  Call Extruder 0.1366
  MoveL (T14464) to (106.09, 106.63, 16.1) mm, rotated rx 180 ry 0 rz -180 deg; joints [1.434, 67.125, -29.697, 2.359, -37.451, -1.873]
  Call Extruder 0.01306
  MoveL (T14465) to (106.44, 106.98, 16.1) mm, rotated rx 180 ry 0 rz -180 deg; joints [1.434, 67.125, -29.697, 2.359, -37.451, -1.873]
  Call Extruder 0.12393
  MoveL (T14466) to (111.15, 106.98, 16.1) mm, rotated rx 180 ry 0 rz -180 deg; joints [1.434, 67.125, -29.697, 2.359, -37.451, -1.873]
  Set speed (150.0 mm/s)
  MoveL (T14467) to (112.51, 106.28, 16.1) mm, rotated rx 180 ry 0 rz -180 deg; joints [1.744, 66.421, -28.373, 2.828, -38.082, -2.227]
  Set speed (25.0 mm/s)
  MoveL (T14468) to (112.51, 106.28, 16.1) mm, rotated rx 180 ry 0 rz -180 deg; joints [1.744, 66.421, -28.373, 2.828, -38.082, -2.227]
  Call Extruder 0.22808
  MoveL (T14469) to (121.19, 106.28, 16.1) mm, rotated rx 180 ry 0 rz -180 deg; joints [1.744, 66.421, -28.373, 2.828, -38.082, -2.227]
  Call Extruder 0.00923
  MoveL (T14470) to (121.19, 106.63, 16.1) mm, rotated rx 180 ry 0 rz -180 deg; joints [1.681, 66.417, -28.365, 2.726, -38.083, -2.146]
  Call Extruder 0.21306
  MoveL (T14471) to (113.08, 106.63, 16.1) mm, rotated rx 180 ry 0 rz -180 deg; joints [1.681, 66.417, -28.365, 2.726, -38.083, -2.146]
  Call Extruder 0.01306
  MoveL (T14472) to (113.43, 106.98, 16.1) mm, rotated rx 180 ry 0 rz -180 deg; joints [1.681, 66.417, -28.365, 2.726, -38.083, -2.146]
  Call Extruder 0.20382
  MoveL (T14473) to (121.19, 106.98, 16.1) mm, rotated rx 180 ry 0 rz -180 deg; joints [1.436, 66.973, -29.411, 2.354, -37.585, -1.866]
  Call Extruder 0.00923
  MoveL (T14474) to (121.19, 107.33, 16.1) mm, rotated rx 180 ry 0 rz -180 deg; joints [1.436, 66.973, -29.411, 2.354, -37.585, -1.866]
  Call Extruder 0.09038
  MoveL (T14475) to (117.75, 107.33, 16.1) mm, rotated rx 180 ry 0 rz -180 deg; joints [1.436, 66.973, -29.411, 2.354, -37.585, -1.866]
  Call Extruder 0.00923
  MoveL (T14476) to (117.75, 107.68, 16.1) mm, rotated rx 180 ry 0 rz -180 deg; joints [1.436, 66.973, -29.411, 2.354, -37.585, -1.866]
  Call Extruder 0.09038
  MoveL (T14477) to (121.19, 107.68, 16.1) mm, rotated rx 180 ry 0 rz -180 deg; joints [1.437, 66.821, -29.126, 2.35, -37.719, -1.859]
  Call Extruder 0.00923
  MoveL (T14478) to (121.19, 108.03, 16.1) mm, rotated rx 180 ry 0 rz -180 deg; joints [1.437, 66.821, -29.126, 2.35, -37.719, -1.859]
  Call Extruder 0.09039
  MoveL (T14479) to (117.75, 108.03, 16.1) mm, rotated rx 180 ry 0 rz -180 deg; joints [1.437, 66.821, -29.126, 2.35, -37.719, -1.859]
  Call Extruder 0.00923
  MoveL (T14480) to (117.75, 108.38, 16.1) mm, rotated rx 180 ry 0 rz -180 deg; joints [1.437, 66.821, -29.126, 2.35, -37.719, -1.859]
  Call Extruder 0.09039
  MoveL (T14481) to (121.19, 108.38, 16.1) mm, rotated rx 180 ry 0 rz -180 deg; joints [1.618, 66.412, -28.357, 2.624, -38.085, -2.066]
  Call Extruder 0.00923
  MoveL (T14482) to (121.19, 108.73, 16.1) mm, rotated rx 180 ry 0 rz -180 deg; joints [1.618, 66.412, -28.357, 2.624, -38.085, -2.066]
  Call Extruder 0.0904
  MoveL (T14483) to (117.75, 108.73, 16.1) mm, rotated rx 180 ry 0 rz -180 deg; joints [1.618, 66.412, -28.357, 2.624, -38.085, -2.066]
  Call Extruder 0.00923
  MoveL (T14484) to (117.75, 109.09, 16.1) mm, rotated rx 180 ry 0 rz -180 deg; joints [1.555, 66.408, -28.349, 2.522, -38.086, -1.985]
  Call Extruder 0.0904
  MoveL (T14485) to (121.19, 109.09, 16.1) mm, rotated rx 180 ry 0 rz -180 deg; joints [1.555, 66.408, -28.349, 2.522, -38.086, -1.985]
  Call Extruder 0.00923
  MoveL (T14486) to (121.19, 109.44, 16.1) mm, rotated rx 180 ry 0 rz -180 deg; joints [1.555, 66.408, -28.349, 2.522, -38.086, -1.985]
  Call Extruder 0.0904
  MoveL (T14487) to (117.75, 109.44, 16.1) mm, rotated rx 180 ry 0 rz -180 deg; joints [1.439, 66.67, -28.842, 2.345, -37.851, -1.852]
  Call Extruder 0.00923
  MoveL (T14488) to (117.75, 109.79, 16.1) mm, rotated rx 180 ry 0 rz -180 deg; joints [1.439, 66.67, -28.842, 2.345, -37.851, -1.852]
  Call Extruder 0.09041
  MoveL (T14489) to (121.19, 109.79, 16.1) mm, rotated rx 180 ry 0 rz -180 deg; joints [1.439, 66.67, -28.842, 2.345, -37.851, -1.852]
  Call Extruder 0.00923
  MoveL (T14490) to (121.19, 110.14, 16.1) mm, rotated rx 180 ry 0 rz -180 deg; joints [1.44, 66.521, -28.56, 2.341, -37.983, -1.845]
  Call Extruder 0.09041
  MoveL (T14491) to (117.75, 110.14, 16.1) mm, rotated rx 180 ry 0 rz -180 deg; joints [1.44, 66.521, -28.56, 2.341, -37.983, -1.845]
  Call Extruder 0.00268
  MoveL (T14492) to (117.75, 110.24, 16.1) mm, rotated rx 180 ry 0 rz -180 deg; joints [1.44, 66.521, -28.56, 2.341, -37.983, -1.845]
  Call Extruder 0.00927
  MoveL (T14493) to (118, 110.49, 16.1) mm, rotated rx 180 ry 0 rz -180 deg; joints [1.512, 66.359, -28.256, 2.45, -38.128, -1.928]
  Call Extruder 0.08386
  MoveL (T14494) to (121.19, 110.49, 16.1) mm, rotated rx 180 ry 0 rz -180 deg; joints [1.512, 66.359, -28.256, 2.45, -38.128, -1.928]
  Call Extruder 0.00923
  MoveL (T14495) to (121.19, 110.84, 16.1) mm, rotated rx 180 ry 0 rz -180 deg; joints [1.512, 66.359, -28.256, 2.45, -38.128, -1.928]
  Call Extruder 0.07462
  MoveL (T14496) to (118.35, 110.84, 16.1) mm, rotated rx 180 ry 0 rz -180 deg; joints [1.512, 66.359, -28.256, 2.45, -38.128, -1.928]
  Call Extruder 0.01306
  MoveL (T14497) to (118.7, 111.19, 16.1) mm, rotated rx 180 ry 0 rz -180 deg; joints [1.512, 66.359, -28.256, 2.45, -38.128, -1.928]
  Call Extruder 0.06539
  MoveL (T14498) to (121.19, 111.19, 16.1) mm, rotated rx 180 ry 0 rz -180 deg; joints [1.512, 66.359, -28.256, 2.45, -38.128, -1.928]
  Call Extruder 0.00923
  MoveL (T14499) to (121.19, 111.55, 16.1) mm, rotated rx 180 ry 0 rz -180 deg; joints [1.512, 66.359, -28.256, 2.45, -38.128, -1.928]
  Call Extruder 0.05615
  MoveL (T14500) to (119.05, 111.55, 16.1) mm, rotated rx 180 ry 0 rz -180 deg; joints [1.512, 66.359, -28.256, 2.45, -38.128, -1.928]
  Call Extruder 0.01306
  MoveL (T14501) to (119.4, 111.9, 16.1) mm, rotated rx 180 ry 0 rz -180 deg; joints [1.512, 66.359, -28.256, 2.45, -38.128, -1.928]
  Call Extruder 0.05101
  MoveL (T14502) to (121.34, 111.9, 16.1) mm, rotated rx 180 ry 0 rz -180 deg; joints [1.512, 66.359, -28.256, 2.45, -38.128, -1.928]
  Set speed (45.0 mm/s)
  Call Extruder -1.6
  MoveL (T14503) to (121.34, 111.9, 16.1) mm, rotated rx 180 ry 0 rz -180 deg; joints [1.44, 66.521, -28.56, 2.341, -37.983, -1.845]
  Set speed (120.0 mm/s)
  MoveL (T14504) to (121.34, 111.9, 16.1) mm, rotated rx 180 ry 0 rz -180 deg; joints [1.44, 66.521, -28.56, 2.341, -37.983, -1.845]
  Call Extruder -0.38
  MoveL (T14505) to (120.28, 111.9, 16.1) mm, rotated rx 180 ry 0 rz -180 deg; joints [1.44, 66.521, -28.56, 2.341, -37.983, -1.845]
  Set speed (45.0 mm/s)
  Call Extruder -0.02
  MoveL (T14506) to (120.28, 111.9, 16.1) mm, rotated rx 180 ry 0 rz -180 deg; joints [1.44, 66.521, -28.56, 2.341, -37.983, -1.845]
  Set speed (150.0 mm/s)
  MoveL (T14507) to (120.28, 111.9, 18.1) mm, rotated rx 180 ry 0 rz -180 deg; joints [1.44, 66.559, -28.633, 2.342, -37.949, -1.847]
  MoveL (T14508) to (120.87, 104.13, 18.1) mm, rotated rx 180 ry 0 rz -180 deg; joints [1.44, 66.559, -28.633, 2.342, -37.949, -1.847]
  MoveL (T14509) to (120.87, 104.13, 16.1) mm, rotated rx 180 ry 0 rz -180 deg; joints [1.44, 66.559, -28.633, 2.342, -37.949, -1.847]
  Set speed (40.0 mm/s)
  Call Extruder 2.0
  MoveL (T14510) to (120.87, 104.13, 16.1) mm, rotated rx 180 ry 0 rz -180 deg; joints [1.44, 66.559, -28.633, 2.342, -37.949, -1.847]
  Set speed (50.0 mm/s)
  MoveL (T14511) to (120.87, 104.13, 16.1) mm, rotated rx 180 ry 0 rz -180 deg; joints [1.44, 66.559, -28.633, 2.342, -37.949, -1.847]
  Call Extruder 0.01219
  MoveL (T14512) to (121.16, 103.84, 16.1) mm, rotated rx 180 ry 0 rz -180 deg; joints [1.44, 66.559, -28.633, 2.342, -37.949, -1.847]
  Set speed (45.0 mm/s)
  Call Extruder -1.6
  MoveL (T14513) to (121.16, 103.84, 16.1) mm, rotated rx 180 ry 0 rz -180 deg; joints [1.44, 66.321, -28.593, 2.352, -37.752, -1.86]
  Set speed (120.0 mm/s)
  MoveL (T14514) to (121.16, 103.84, 16.1) mm, rotated rx 180 ry 0 rz -180 deg; joints [1.407, 66.288, -28.531, 2.298, -37.78, -1.816]
  Call Extruder -0.14257
  MoveL (T14515) to (120.87, 104.13, 16.1) mm, rotated rx 180 ry 0 rz -180 deg; joints [1.407, 66.502, -28.567, 2.288, -37.958, -1.805]
  Set speed (45.0 mm/s)
  Call Extruder -0.25743
  MoveL (T14516) to (120.87, 104.13, 16.1) mm, rotated rx 180 ry 0 rz -180 deg; joints [1.407, 66.502, -28.567, 2.288, -37.958, -1.805]
  Set speed (150.0 mm/s)
  MoveL (T14517) to (120.87, 104.13, 18.1) mm, rotated rx 180 ry 0 rz -180 deg; joints [1.407, 66.502, -28.567, 2.288, -37.958, -1.805]
  MoveL (T14518) to (104.34, 103.54, 18.1) mm, rotated rx 180 ry 0 rz -180 deg; joints [1.407, 66.502, -28.567, 2.288, -37.958, -1.805]
  MoveL (T14519) to (104.34, 103.54, 16.3) mm, rotated rx 180 ry 0 rz -180 deg; joints [1.407, 66.502, -28.567, 2.288, -37.958, -1.805]
  Set speed (40.0 mm/s)
  Call Extruder 2.0
  MoveL (T14520) to (104.34, 103.54, 16.3) mm, rotated rx 180 ry 0 rz -180 deg; joints [1.407, 66.502, -28.567, 2.288, -37.958, -1.805]
  Call Extruder 0.52159
  MoveL (T14521) to (121.46, 103.54, 16.3) mm, rotated rx 180 ry 0 rz -180 deg; joints [1.407, 66.502, -28.567, 2.288, -37.958, -1.805]
  Call Extruder 0.54596
  MoveL (T14522) to (121.46, 121.46, 16.3) mm, rotated rx 180 ry 0 rz -180 deg; joints [1.363, 71.341, -37.668, 2.458, -33.696, -2.045]
  Call Extruder 0.54596
  MoveL (T14523) to (103.54, 121.46, 16.3) mm, rotated rx 180 ry 0 rz -180 deg; joints [1.363, 71.341, -37.668, 2.458, -33.696, -2.045]
  Call Extruder 0.54596
  MoveL (T14524) to (103.54, 103.54, 16.3) mm, rotated rx 180 ry 0 rz -180 deg; joints [1.363, 71.341, -37.668, 2.458, -33.696, -2.045]
  Call Extruder 0.02254
  MoveL (T14525) to (104.28, 103.54, 16.3) mm, rotated rx 180 ry 0 rz -180 deg; joints [3.241, 71.568, -38.096, 5.863, -33.61, -4.888]
  Set speed (150.0 mm/s)
  MoveL (T14526) to (103.53, 103.13, 16.3) mm, rotated rx 180 ry 0 rz -180 deg; joints [3.241, 71.568, -38.096, 5.863, -33.61, -4.888]
  Set speed (40.0 mm/s)
  MoveL (T14527) to (103.53, 103.13, 16.3) mm, rotated rx 180 ry 0 rz -180 deg; joints [3.241, 71.568, -38.096, 5.863, -33.61, -4.888]
  Call Extruder 0.55858
  MoveL (T14528) to (121.87, 103.13, 16.3) mm, rotated rx 180 ry 0 rz -180 deg; joints [3.241, 71.568, -38.096, 5.863, -33.61, -4.888]
  Call Extruder 0.57077
  MoveL (T14529) to (121.87, 121.87, 16.3) mm, rotated rx 180 ry 0 rz -180 deg; joints [3.351, 66.488, -28.54, 5.439, -38.073, -4.287]
  Call Extruder 0.57077
  MoveL (T14530) to (103.13, 121.87, 16.3) mm, rotated rx 180 ry 0 rz -180 deg; joints [3.351, 66.488, -28.54, 5.439, -38.073, -4.287]
  Call Extruder 0.57077
  MoveL (T14531) to (103.13, 103.13, 16.3) mm, rotated rx 180 ry 0 rz -180 deg; joints [3.351, 66.488, -28.54, 5.439, -38.073, -4.287]
  Call Extruder 0.01036
  MoveL (T14532) to (103.47, 103.13, 16.3) mm, rotated rx 180 ry 0 rz -180 deg; joints [1.409, 66.297, -28.181, 2.283, -38.138, -1.796]
  Set speed (150.0 mm/s)
  MoveL (T14533) to (102.72, 102.81, 16.3) mm, rotated rx 180 ry 0 rz -180 deg; joints [1.409, 66.297, -28.181, 2.283, -38.138, -1.796]
  Set speed (25.0 mm/s)
  MoveL (T14534) to (102.72, 102.81, 16.3) mm, rotated rx 180 ry 0 rz -180 deg; joints [1.409, 66.297, -28.181, 2.283, -38.138, -1.796]
  Call Extruder 0.00259
  MoveL (T14535) to (102.72, 102.72, 16.3) mm, rotated rx 180 ry 0 rz -180 deg; joints [1.407, 66.487, -28.538, 2.288, -37.971, -1.804]
  Call Extruder 0.59557
  MoveL (T14536) to (122.28, 102.72, 16.3) mm, rotated rx 180 ry 0 rz -180 deg; joints [1.407, 66.487, -28.538, 2.288, -37.971, -1.804]
  Call Extruder 0.59557
  MoveL (T14537) to (122.28, 122.28, 16.3) mm, rotated rx 180 ry 0 rz -180 deg; joints [1.407, 66.487, -28.538, 2.288, -37.971, -1.804]
  Call Extruder 0.59557
  MoveL (T14538) to (102.72, 122.28, 16.3) mm, rotated rx 180 ry 0 rz -180 deg; joints [1.365, 66.293, -28.173, 2.211, -38.141, -1.739]
  Call Extruder 0.59115
  MoveL (T14539) to (102.72, 102.87, 16.3) mm, rotated rx 180 ry 0 rz -180 deg; joints [1.365, 66.293, -28.173, 2.211, -38.141, -1.739]
  Set speed (150.0 mm/s)
  MoveL (T14540) to (102.78, 102.75, 16.3) mm, rotated rx 180 ry 0 rz -180 deg; joints [1.365, 66.293, -28.173, 2.211, -38.141, -1.739]
  Set speed (45.0 mm/s)
  Call Extruder -1.6
  MoveL (T14541) to (102.78, 102.75, 16.3) mm, rotated rx 180 ry 0 rz -180 deg; joints [1.365, 66.293, -28.173, 2.211, -38.141, -1.739]
  Set speed (120.0 mm/s)
  MoveL (T14542) to (102.78, 102.75, 16.3) mm, rotated rx 180 ry 0 rz -180 deg; joints [1.365, 66.293, -28.173, 2.211, -38.141, -1.739]
  Call Extruder -0.05166
  MoveL (T14543) to (102.72, 102.72, 16.3) mm, rotated rx 180 ry 0 rz -180 deg; joints [1.365, 66.293, -28.173, 2.211, -38.141, -1.739]
  Call Extruder -0.32834
  MoveL (T14544) to (103.65, 102.72, 16.3) mm, rotated rx 180 ry 0 rz -180 deg; joints [1.319, 71.466, -37.904, 2.386, -33.585, -1.988]
  Set speed (45.0 mm/s)
  Call Extruder -0.02
  MoveL (T14545) to (103.65, 102.72, 16.3) mm, rotated rx 180 ry 0 rz -180 deg; joints [1.319, 71.466, -37.904, 2.386, -33.585, -1.988]
  Set speed (150.0 mm/s)
  MoveL (T14546) to (103.65, 102.72, 18.3) mm, rotated rx 180 ry 0 rz -180 deg; joints [3.282, 71.704, -38.353, 5.954, -33.494, -4.971]
  MoveL (T14547) to (103.84, 106.29, 18.3) mm, rotated rx 180 ry 0 rz -180 deg; joints [3.282, 71.704, -38.353, 5.954, -33.494, -4.971]
  MoveL (T14548) to (103.84, 106.29, 16.3) mm, rotated rx 180 ry 0 rz -180 deg; joints [3.398, 66.39, -28.356, 5.504, -38.163, -4.333]
  Set speed (40.0 mm/s)
  Call Extruder 2.0
  MoveL (T14549) to (103.84, 106.29, 16.3) mm, rotated rx 180 ry 0 rz -180 deg; joints [1.366, 66.191, -27.981, 2.208, -38.23, -1.735]
  Set speed (42.3 mm/s)
  MoveL (T14550) to (103.84, 106.29, 16.3) mm, rotated rx 180 ry 0 rz -180 deg; joints [1.366, 66.191, -27.981, 2.208, -38.23, -1.735]
  Call Extruder 0.07441
  MoveL (T14551) to (103.84, 103.84, 16.3) mm, rotated rx 180 ry 0 rz -180 deg; joints [1.365, 66.278, -28.144, 2.211, -38.154, -1.739]
  Call Extruder 0.0111
  MoveL (T14552) to (104.1, 104.1, 16.3) mm, rotated rx 180 ry 0 rz -180 deg; joints [1.365, 66.278, -28.144, 2.211, -38.154, -1.739]
  Call Extruder 0.05294
  MoveL (T14553) to (104.1, 105.84, 16.3) mm, rotated rx 180 ry 0 rz -180 deg; joints [1.365, 66.278, -28.144, 2.211, -38.154, -1.739]
  Call Extruder 0.00661
  MoveL (T14554) to (104.18, 106.04, 16.3) mm, rotated rx 180 ry 0 rz -180 deg; joints [1.332, 66.086, -27.783, 2.149, -38.322, -1.686]
  Call Extruder 0.02065
  MoveL (T14555) to (104.66, 106.52, 16.3) mm, rotated rx 180 ry 0 rz -180 deg; joints [1.332, 66.086, -27.783, 2.149, -38.322, -1.686]
  Call Extruder 0.03528
  MoveL (T14556) to (103.84, 107.34, 16.3) mm, rotated rx 180 ry 0 rz -180 deg; joints [1.332, 66.086, -27.783, 2.149, -38.322, -1.686]
  Call Extruder 0.03385
  MoveL (T14557) to (103.84, 108.45, 16.3) mm, rotated rx 180 ry 0 rz -180 deg; joints [1.332, 66.086, -27.783, 2.149, -38.322, -1.686]
  Call Extruder 0.54738
  MoveL (T14558) to (116.55, 121.16, 16.3) mm, rotated rx 180 ry 0 rz -180 deg; joints [1.323, 66.085, -27.782, 2.134, -38.322, -1.675]
  Call Extruder 0.03385
  MoveL (T14559) to (117.66, 121.16, 16.3) mm, rotated rx 180 ry 0 rz -180 deg; joints [1.323, 66.085, -27.782, 2.134, -38.322, -1.675]
  Call Extruder 0.05922
  MoveL (T14560) to (119.04, 119.78, 16.3) mm, rotated rx 180 ry 0 rz -180 deg; joints [1.323, 66.085, -27.782, 2.134, -38.322, -1.675]
  Call Extruder 0.00883
  MoveL (T14561) to (119.24, 119.99, 16.3) mm, rotated rx 180 ry 0 rz -180 deg; joints [1.276, 71.591, -38.14, 2.314, -33.472, -1.93]
  Call Extruder 0.02274
  MoveL (T14562) to (119.99, 119.99, 16.3) mm, rotated rx 180 ry 0 rz -180 deg; joints [1.276, 71.591, -38.14, 2.314, -33.472, -1.93]
  Call Extruder 0.05034
  MoveL (T14563) to (121.16, 121.16, 16.3) mm, rotated rx 180 ry 0 rz -180 deg; joints [3.322, 71.842, -38.612, 6.046, -33.377, -5.054]
  Call Extruder 0.07441
  MoveL (T14564) to (118.71, 121.16, 16.3) mm, rotated rx 180 ry 0 rz -180 deg; joints [3.322, 71.842, -38.612, 6.046, -33.377, -5.054]
  Set speed (45.0 mm/s)
  Call Extruder -1.6
  MoveL (T14565) to (118.71, 121.16, 16.3) mm, rotated rx 180 ry 0 rz -180 deg; joints [3.322, 71.842, -38.612, 6.046, -33.377, -5.054]
  Set speed (120.0 mm/s)
  MoveL (T14566) to (118.71, 121.16, 16.3) mm, rotated rx 180 ry 0 rz -180 deg; joints [3.445, 66.292, -28.172, 5.569, -38.252, -4.379]
  Call Extruder -0.38
  MoveL (T14567) to (119.78, 121.16, 16.3) mm, rotated rx 180 ry 0 rz -180 deg; joints [3.445, 66.292, -28.172, 5.569, -38.252, -4.379]
  Set speed (45.0 mm/s)
  Call Extruder -0.02
  MoveL (T14568) to (119.78, 121.16, 16.3) mm, rotated rx 180 ry 0 rz -180 deg; joints [3.445, 66.292, -28.172, 5.569, -38.252, -4.379]
  Set speed (150.0 mm/s)
  MoveL (T14569) to (119.78, 121.16, 18.3) mm, rotated rx 180 ry 0 rz -180 deg; joints [1.339, 66.086, -27.784, 2.16, -38.322, -1.695]
  MoveL (T14570) to (117.37, 115.49, 18.3) mm, rotated rx 180 ry 0 rz -180 deg; joints [1.339, 66.086, -27.784, 2.16, -38.322, -1.695]
  MoveL (T14571) to (117.37, 115.49, 16.3) mm, rotated rx 180 ry 0 rz -180 deg; joints [1.339, 66.086, -27.784, 2.16, -38.322, -1.695]
  Set speed (40.0 mm/s)
  Call Extruder 2.0
  MoveL (T14572) to (117.37, 115.49, 16.3) mm, rotated rx 180 ry 0 rz -180 deg; joints [1.339, 66.086, -27.784, 2.16, -38.322, -1.695]
  Set speed (42.3 mm/s)
  MoveL (T14573) to (117.37, 115.49, 16.3) mm, rotated rx 180 ry 0 rz -180 deg; joints [1.326, 66.1, -27.811, 2.139, -38.309, -1.679]
  Call Extruder 0.05347
  MoveL (T14574) to (117.37, 113.73, 16.3) mm, rotated rx 180 ry 0 rz -180 deg; joints [1.326, 66.1, -27.811, 2.139, -38.309, -1.679]
  Call Extruder 0.02094
  MoveL (T14575) to (117.86, 113.25, 16.3) mm, rotated rx 180 ry 0 rz -180 deg; joints [1.326, 66.1, -27.811, 2.139, -38.309, -1.679]
  Call Extruder 0.2558
  MoveL (T14576) to (111.92, 107.31, 16.3) mm, rotated rx 180 ry 0 rz -180 deg; joints [1.326, 66.1, -27.811, 2.139, -38.309, -1.679]
  Call Extruder 0.01143
  MoveL (T14577) to (112.18, 107.05, 16.3) mm, rotated rx 180 ry 0 rz -180 deg; joints [1.326, 66.1, -27.811, 2.139, -38.309, -1.679]
  Call Extruder 0.02508
  MoveL (T14578) to (112.77, 107.63, 16.3) mm, rotated rx 180 ry 0 rz -180 deg; joints [1.326, 66.1, -27.811, 2.139, -38.309, -1.679]
  Call Extruder 0.38433
  MoveL (T14579) to (103.84, 116.55, 16.3) mm, rotated rx 180 ry 0 rz -180 deg; joints [1.326, 66.1, -27.811, 2.139, -38.309, -1.679]
  Call Extruder 0.03385
  MoveL (T14580) to (103.84, 117.66, 16.3) mm, rotated rx 180 ry 0 rz -180 deg; joints [1.326, 66.1, -27.811, 2.139, -38.309, -1.679]
  Call Extruder 0.15054
  MoveL (T14581) to (107.34, 121.16, 16.3) mm, rotated rx 180 ry 0 rz -180 deg; joints [1.326, 66.1, -27.811, 2.139, -38.309, -1.679]
  Call Extruder 0.03385
  MoveL (T14582) to (108.45, 121.16, 16.3) mm, rotated rx 180 ry 0 rz -180 deg; joints [1.326, 66.1, -27.811, 2.139, -38.309, -1.679]
  Call Extruder 0.40697
  MoveL (T14583) to (117.9, 111.71, 16.3) mm, rotated rx 180 ry 0 rz -180 deg; joints [1.326, 66.1, -27.811, 2.139, -38.309, -1.679]
  Call Extruder 0.04304
  MoveL (T14584) to (116.9, 110.71, 16.3) mm, rotated rx 180 ry 0 rz -180 deg; joints [1.323, 66.085, -27.782, 2.134, -38.322, -1.675]
  Call Extruder 0.00661
  MoveL (T14585) to (116.81, 110.51, 16.3) mm, rotated rx 180 ry 0 rz -180 deg; joints [1.323, 66.085, -27.782, 2.134, -38.322, -1.675]
  Call Extruder 0.07083
  MoveL (T14586) to (116.81, 108.19, 16.3) mm, rotated rx 180 ry 0 rz -180 deg; joints [1.323, 66.085, -27.782, 2.134, -38.322, -1.675]
  Call Extruder 0.55882
  MoveL (T14587) to (103.84, 121.16, 16.3) mm, rotated rx 180 ry 0 rz -180 deg; joints [1.321, 66.32, -28.224, 2.14, -38.116, -1.684]
  Call Extruder 0.07441
  MoveL (T14588) to (106.29, 121.16, 16.3) mm, rotated rx 180 ry 0 rz -180 deg; joints [1.321, 66.32, -28.224, 2.14, -38.116, -1.684]
  Set speed (45.0 mm/s)
  Call Extruder -1.6
  MoveL (T14589) to (106.29, 121.16, 16.3) mm, rotated rx 180 ry 0 rz -180 deg; joints [1.321, 66.32, -28.224, 2.14, -38.116, -1.684]
  Set speed (120.0 mm/s)
  MoveL (T14590) to (106.29, 121.16, 16.3) mm, rotated rx 180 ry 0 rz -180 deg; joints [1.321, 66.32, -28.224, 2.14, -38.116, -1.684]
  Call Extruder -0.38
  MoveL (T14591) to (105.22, 121.16, 16.3) mm, rotated rx 180 ry 0 rz -180 deg; joints [1.321, 66.32, -28.224, 2.14, -38.116, -1.684]
  Set speed (45.0 mm/s)
  Call Extruder -0.02
  MoveL (T14592) to (105.22, 121.16, 16.3) mm, rotated rx 180 ry 0 rz -180 deg; joints [1.321, 66.32, -28.224, 2.14, -38.116, -1.684]
  Set speed (150.0 mm/s)
  MoveL (T14593) to (105.22, 121.16, 18.3) mm, rotated rx 180 ry 0 rz -180 deg; joints [1.321, 66.32, -28.224, 2.14, -38.116, -1.684]
  MoveL (T14594) to (103.84, 115.5, 18.3) mm, rotated rx 180 ry 0 rz -180 deg; joints [1.321, 66.082, -28.184, 2.15, -37.917, -1.696]
  MoveL (T14595) to (103.84, 115.5, 16.3) mm, rotated rx 180 ry 0 rz -180 deg; joints [1.378, 70.81, -37.065, 2.48, -33.769, -2.062]
  Set speed (40.0 mm/s)
  Call Extruder 2.0
  MoveL (T14596) to (103.84, 115.5, 16.3) mm, rotated rx 180 ry 0 rz -180 deg; joints [1.378, 71.045, -37.112, 2.468, -33.958, -2.048]
  Set speed (42.3 mm/s)
  MoveL (T14597) to (103.84, 115.5, 16.3) mm, rotated rx 180 ry 0 rz -180 deg; joints [1.378, 71.045, -37.112, 2.468, -33.958, -2.048]
  Call Extruder 0.07441
  MoveL (T14598) to (103.84, 113.06, 16.3) mm, rotated rx 180 ry 0 rz -180 deg; joints [1.378, 71.045, -37.112, 2.468, -33.958, -2.048]
  Call Extruder 0.34896
  MoveL (T14599) to (111.94, 121.16, 16.3) mm, rotated rx 180 ry 0 rz -180 deg; joints [1.378, 71.045, -37.112, 2.468, -33.958, -2.048]
  Call Extruder 0.03385
  MoveL (T14600) to (113.06, 121.16, 16.3) mm, rotated rx 180 ry 0 rz -180 deg; joints [1.378, 71.045, -37.112, 2.468, -33.958, -2.048]
  Call Extruder 0.18576
  MoveL (T14601) to (117.37, 116.84, 16.3) mm, rotated rx 180 ry 0 rz -180 deg; joints [1.378, 71.045, -37.112, 2.468, -33.958, -2.048]
  Call Extruder 0.01595
  MoveL (T14602) to (117.37, 117.37, 16.3) mm, rotated rx 180 ry 0 rz -180 deg; joints [1.445, 71.251, -37.5, 2.599, -33.778, -2.161]
  Call Extruder 0.39664
  MoveL (T14603) to (108.16, 108.16, 16.3) mm, rotated rx 180 ry 0 rz -180 deg; joints [1.445, 71.251, -37.5, 2.599, -33.778, -2.161]
  Call Extruder 0.01622
  MoveL (T14604) to (107.63, 108.16, 16.3) mm, rotated rx 180 ry 0 rz -180 deg; joints [1.506, 71.256, -37.509, 2.709, -33.776, -2.252]
  Call Extruder 0.16301
  MoveL (T14605) to (103.84, 111.94, 16.3) mm, rotated rx 180 ry 0 rz -180 deg; joints [1.506, 71.256, -37.509, 2.709, -33.776, -2.252]
  Call Extruder 0.07441
  MoveL (T14606) to (103.84, 109.5, 16.3) mm, rotated rx 180 ry 0 rz -180 deg; joints [1.399, 70.923, -36.883, 2.498, -34.065, -2.069]
  Set speed (45.0 mm/s)
  Call Extruder -1.6
  MoveL (T14607) to (103.84, 109.5, 16.3) mm, rotated rx 180 ry 0 rz -180 deg; joints [1.399, 70.923, -36.883, 2.498, -34.065, -2.069]
  Set speed (120.0 mm/s)
  MoveL (T14608) to (103.84, 109.5, 16.3) mm, rotated rx 180 ry 0 rz -180 deg; joints [1.399, 70.923, -36.883, 2.498, -34.065, -2.069]
  Call Extruder -0.38
  MoveL (T14609) to (103.84, 110.57, 16.3) mm, rotated rx 180 ry 0 rz -180 deg; joints [1.4, 70.745, -36.548, 2.49, -34.222, -2.059]
  Set speed (45.0 mm/s)
  Call Extruder -0.02
  MoveL (T14610) to (103.84, 110.57, 16.3) mm, rotated rx 180 ry 0 rz -180 deg; joints [1.567, 71.261, -37.518, 2.819, -33.775, -2.344]
  Set speed (150.0 mm/s)
  MoveL (T14611) to (103.84, 110.57, 18.3) mm, rotated rx 180 ry 0 rz -180 deg; joints [1.567, 71.261, -37.518, 2.819, -33.775, -2.344]
  MoveL (T14612) to (121.17, 112.08, 18.3) mm, rotated rx 180 ry 0 rz -180 deg; joints [1.628, 71.266, -37.527, 2.929, -33.773, -2.435]
  MoveL (T14613) to (121.17, 112.08, 16.3) mm, rotated rx 180 ry 0 rz -180 deg; joints [1.628, 71.266, -37.527, 2.929, -33.773, -2.435]
  Set speed (40.0 mm/s)
  Call Extruder 2.0
  MoveL (T14614) to (121.17, 112.08, 16.3) mm, rotated rx 180 ry 0 rz -180 deg; joints [1.628, 71.266, -37.527, 2.929, -33.773, -2.435]
  Set speed (25.0 mm/s)
  MoveL (T14615) to (121.17, 112.08, 16.3) mm, rotated rx 180 ry 0 rz -180 deg; joints [1.402, 70.568, -36.216, 2.483, -34.378, -2.05]
  Call Extruder 0.21348
  MoveL (T14616) to (121.17, 119.61, 16.3) mm, rotated rx 180 ry 0 rz -180 deg; joints [1.402, 70.568, -36.216, 2.483, -34.378, -2.05]
  Call Extruder 0.01074
  MoveL (T14617) to (120.79, 119.61, 16.3) mm, rotated rx 180 ry 0 rz -180 deg; joints [1.403, 70.393, -35.886, 2.476, -34.532, -2.04]
  Call Extruder 0.20906
  MoveL (T14618) to (120.79, 112.24, 16.3) mm, rotated rx 180 ry 0 rz -180 deg; joints [1.403, 70.393, -35.886, 2.476, -34.532, -2.04]
  Call Extruder 0.01074
  MoveL (T14619) to (120.41, 112.24, 16.3) mm, rotated rx 180 ry 0 rz -180 deg; joints [1.403, 70.393, -35.886, 2.476, -34.532, -2.04]
  Call Extruder 0.20906
  MoveL (T14620) to (120.41, 119.61, 16.3) mm, rotated rx 180 ry 0 rz -180 deg; joints [1.689, 71.271, -37.537, 3.039, -33.771, -2.527]
  Call Extruder 0.01074
  MoveL (T14621) to (120.03, 119.61, 16.3) mm, rotated rx 180 ry 0 rz -180 deg; joints [1.689, 71.271, -37.537, 3.039, -33.771, -2.527]
  Call Extruder 0.20906
  MoveL (T14622) to (120.03, 112.24, 16.3) mm, rotated rx 180 ry 0 rz -180 deg; joints [1.689, 71.271, -37.537, 3.039, -33.771, -2.527]
  Call Extruder 0.01074
  MoveL (T14623) to (119.65, 112.24, 16.3) mm, rotated rx 180 ry 0 rz -180 deg; joints [1.689, 71.271, -37.537, 3.039, -33.771, -2.527]
  Call Extruder 0.20906
  MoveL (T14624) to (119.65, 119.61, 16.3) mm, rotated rx 180 ry 0 rz -180 deg; joints [1.75, 71.276, -37.548, 3.149, -33.769, -2.618]
  Call Extruder 0.00729
  MoveL (T14625) to (119.4, 119.61, 16.3) mm, rotated rx 180 ry 0 rz -180 deg; joints [1.75, 71.276, -37.548, 3.149, -33.769, -2.618]
  Call Extruder 0.00489
  MoveL (T14626) to (119.28, 119.49, 16.3) mm, rotated rx 180 ry 0 rz -180 deg; joints [1.405, 70.219, -35.559, 2.469, -34.685, -2.03]
  Call Extruder 0.20197
  MoveL (T14627) to (119.28, 112.36, 16.3) mm, rotated rx 180 ry 0 rz -180 deg; joints [1.405, 70.219, -35.559, 2.469, -34.685, -2.03]
  Call Extruder 0.01518
  MoveL (T14628) to (118.9, 112.74, 16.3) mm, rotated rx 180 ry 0 rz -180 deg; joints [1.405, 70.219, -35.559, 2.469, -34.685, -2.03]
  Call Extruder 0.18048
  MoveL (T14629) to (118.9, 119.11, 16.3) mm, rotated rx 180 ry 0 rz -180 deg; joints [1.406, 70.047, -35.234, 2.462, -34.837, -2.021]
  Call Extruder 0.0152
  MoveL (T14630) to (118.52, 118.73, 16.3) mm, rotated rx 180 ry 0 rz -180 deg; joints [1.406, 70.047, -35.234, 2.462, -34.837, -2.021]
  Call Extruder 0.159
  MoveL (T14631) to (118.52, 113.12, 16.3) mm, rotated rx 180 ry 0 rz -180 deg; joints [1.406, 70.047, -35.234, 2.462, -34.837, -2.021]
  Call Extruder 0.01518
  MoveL (T14632) to (118.14, 113.5, 16.3) mm, rotated rx 180 ry 0 rz -180 deg; joints [1.811, 71.282, -37.558, 3.259, -33.767, -2.71]
  Call Extruder 0.13752
  MoveL (T14633) to (118.14, 118.35, 16.3) mm, rotated rx 180 ry 0 rz -180 deg; joints [1.811, 71.282, -37.558, 3.259, -33.767, -2.71]
  Call Extruder 0.0152
  MoveL (T14634) to (117.76, 117.97, 16.3) mm, rotated rx 180 ry 0 rz -180 deg; joints [1.811, 71.282, -37.558, 3.259, -33.767, -2.71]
  Call Extruder 0.12227
  MoveL (T14635) to (117.76, 113.66, 16.3) mm, rotated rx 180 ry 0 rz -180 deg; joints [1.871, 71.288, -37.569, 3.369, -33.764, -2.801]
  Set speed (45.0 mm/s)
  Call Extruder -1.6
  MoveL (T14636) to (117.76, 113.66, 16.3) mm, rotated rx 180 ry 0 rz -180 deg; joints [1.871, 71.288, -37.569, 3.369, -33.764, -2.801]
  Set speed (120.0 mm/s)
  MoveL (T14637) to (117.76, 113.66, 16.3) mm, rotated rx 180 ry 0 rz -180 deg; joints [1.408, 69.875, -34.912, 2.455, -34.988, -2.012]
  Call Extruder -0.38
  MoveL (T14638) to (117.76, 114.72, 16.3) mm, rotated rx 180 ry 0 rz -180 deg; joints [1.408, 69.875, -34.912, 2.455, -34.988, -2.012]
  Set speed (45.0 mm/s)
  Call Extruder -0.02
  MoveL (T14639) to (117.76, 114.72, 16.3) mm, rotated rx 180 ry 0 rz -180 deg; joints [1.409, 69.705, -34.592, 2.449, -35.138, -2.003]
  Set speed (150.0 mm/s)
  MoveL (T14640) to (117.76, 114.72, 18.3) mm, rotated rx 180 ry 0 rz -180 deg; joints [1.409, 69.705, -34.592, 2.449, -35.138, -2.003]
  MoveL (T14641) to (121.34, 104.69, 18.3) mm, rotated rx 180 ry 0 rz -180 deg; joints [1.932, 71.294, -37.581, 3.479, -33.762, -2.893]
  MoveL (T14642) to (121.34, 104.69, 16.3) mm, rotated rx 180 ry 0 rz -180 deg; joints [1.932, 71.294, -37.581, 3.479, -33.762, -2.893]
  Set speed (40.0 mm/s)
  Call Extruder 2.0
  MoveL (T14643) to (121.34, 104.69, 16.3) mm, rotated rx 180 ry 0 rz -180 deg; joints [1.932, 71.294, -37.581, 3.479, -33.762, -2.893]
  Call Extruder 0.03095
  MoveL (T14644) to (120.62, 103.98, 16.3) mm, rotated rx 180 ry 0 rz -180 deg; joints [1.932, 71.294, -37.581, 3.479, -33.762, -2.893]
  Call Extruder 0.01768
  MoveL (T14645) to (120.05, 103.98, 16.3) mm, rotated rx 180 ry 0 rz -180 deg; joints [1.932, 71.294, -37.581, 3.479, -33.762, -2.893]
  Call Extruder 0.04803
  MoveL (T14646) to (121.16, 105.09, 16.3) mm, rotated rx 180 ry 0 rz -180 deg; joints [1.993, 71.3, -37.592, 3.589, -33.76, -2.985]
  Call Extruder 0.01769
  MoveL (T14647) to (121.16, 105.67, 16.3) mm, rotated rx 180 ry 0 rz -180 deg; joints [1.993, 71.3, -37.592, 3.589, -33.76, -2.985]
  Call Extruder 0.07889
  MoveL (T14648) to (119.33, 103.84, 16.3) mm, rotated rx 180 ry 0 rz -180 deg; joints [1.411, 69.536, -34.274, 2.442, -35.287, -1.994]
  Call Extruder 0.01769
  MoveL (T14649) to (118.75, 103.84, 16.3) mm, rotated rx 180 ry 0 rz -180 deg; joints [1.411, 69.536, -34.274, 2.442, -35.287, -1.994]
  Call Extruder 0.10391
  MoveL (T14650) to (121.16, 106.25, 16.3) mm, rotated rx 180 ry 0 rz -180 deg; joints [1.411, 69.536, -34.274, 2.442, -35.287, -1.994]
  Call Extruder 0.01769
  MoveL (T14651) to (121.16, 106.82, 16.3) mm, rotated rx 180 ry 0 rz -180 deg; joints [1.411, 69.536, -34.274, 2.442, -35.287, -1.994]
  Call Extruder 0.12893
  MoveL (T14652) to (118.18, 103.84, 16.3) mm, rotated rx 180 ry 0 rz -180 deg; joints [1.412, 69.369, -33.958, 2.436, -35.435, -1.985]
  Call Extruder 0.01769
  MoveL (T14653) to (117.6, 103.84, 16.3) mm, rotated rx 180 ry 0 rz -180 deg; joints [1.412, 69.369, -33.958, 2.436, -35.435, -1.985]
  Call Extruder 0.15395
  MoveL (T14654) to (121.16, 107.4, 16.3) mm, rotated rx 180 ry 0 rz -180 deg; joints [2.054, 71.306, -37.604, 3.699, -33.757, -3.076]
  Call Extruder 0.01769
  MoveL (T14655) to (121.16, 107.98, 16.3) mm, rotated rx 180 ry 0 rz -180 deg; joints [2.054, 71.306, -37.604, 3.699, -33.757, -3.076]
  Call Extruder 0.17896
  MoveL (T14656) to (117.02, 103.84, 16.3) mm, rotated rx 180 ry 0 rz -180 deg; joints [2.054, 71.306, -37.604, 3.699, -33.757, -3.076]
  Call Extruder 0.01769
  MoveL (T14657) to (116.44, 103.84, 16.3) mm, rotated rx 180 ry 0 rz -180 deg; joints [2.115, 71.313, -37.617, 3.809, -33.755, -3.168]
  Call Extruder 0.20398
  MoveL (T14658) to (121.16, 108.56, 16.3) mm, rotated rx 180 ry 0 rz -180 deg; joints [2.115, 71.313, -37.617, 3.809, -33.755, -3.168]
  Call Extruder 0.01769
  MoveL (T14659) to (121.16, 109.14, 16.3) mm, rotated rx 180 ry 0 rz -180 deg; joints [2.115, 71.313, -37.617, 3.809, -33.755, -3.168]
  Call Extruder 0.229
  MoveL (T14660) to (115.86, 103.84, 16.3) mm, rotated rx 180 ry 0 rz -180 deg; joints [1.414, 69.202, -33.645, 2.43, -35.582, -1.977]
  Call Extruder 0.01769
  MoveL (T14661) to (115.28, 103.84, 16.3) mm, rotated rx 180 ry 0 rz -180 deg; joints [1.414, 69.202, -33.645, 2.43, -35.582, -1.977]
  Call Extruder 0.25402
  MoveL (T14662) to (121.16, 109.72, 16.3) mm, rotated rx 180 ry 0 rz -180 deg; joints [1.415, 69.037, -33.334, 2.424, -35.727, -1.968]
  Call Extruder 0.01769
  MoveL (T14663) to (121.16, 110.29, 16.3) mm, rotated rx 180 ry 0 rz -180 deg; joints [1.415, 69.037, -33.334, 2.424, -35.727, -1.968]
  Call Extruder 0.27904
  MoveL (T14664) to (114.71, 103.84, 16.3) mm, rotated rx 180 ry 0 rz -180 deg; joints [2.176, 71.32, -37.63, 3.919, -33.752, -3.26]
  Call Extruder 0.01769
  MoveL (T14665) to (114.13, 103.84, 16.3) mm, rotated rx 180 ry 0 rz -180 deg; joints [2.176, 71.32, -37.63, 3.919, -33.752, -3.26]
  Call Extruder 0.30406
  MoveL (T14666) to (121.16, 110.87, 16.3) mm, rotated rx 180 ry 0 rz -180 deg; joints [2.176, 71.32, -37.63, 3.919, -33.752, -3.26]
  Call Extruder 0.01769
  MoveL (T14667) to (121.16, 111.45, 16.3) mm, rotated rx 180 ry 0 rz -180 deg; joints [2.237, 71.327, -37.643, 4.029, -33.75, -3.352]
  Call Extruder 0.32908
  MoveL (T14668) to (113.55, 103.84, 16.3) mm, rotated rx 180 ry 0 rz -180 deg; joints [2.237, 71.327, -37.643, 4.029, -33.75, -3.352]
  Call Extruder 0.01769
  MoveL (T14669) to (112.97, 103.84, 16.3) mm, rotated rx 180 ry 0 rz -180 deg; joints [1.417, 68.872, -33.024, 2.418, -35.872, -1.96]
  Call Extruder 0.3469
  MoveL (T14670) to (120.99, 111.86, 16.3) mm, rotated rx 180 ry 0 rz -180 deg; joints [1.417, 68.872, -33.024, 2.418, -35.872, -1.96]
  Call Extruder 0.01771
  MoveL (T14671) to (120.41, 111.86, 16.3) mm, rotated rx 180 ry 0 rz -180 deg; joints [1.418, 68.709, -32.717, 2.413, -36.016, -1.952]
  Call Extruder 0.13794
  MoveL (T14672) to (117.22, 108.67, 16.3) mm, rotated rx 180 ry 0 rz -180 deg; joints [1.418, 68.709, -32.717, 2.413, -36.016, -1.952]
  Call Extruder 0.01768
  MoveL (T14673) to (117.22, 109.25, 16.3) mm, rotated rx 180 ry 0 rz -180 deg; joints [2.298, 71.334, -37.656, 4.139, -33.747, -3.444]
  Call Extruder 0.1129
  MoveL (T14674) to (119.83, 111.86, 16.3) mm, rotated rx 180 ry 0 rz -180 deg; joints [2.298, 71.334, -37.656, 4.139, -33.747, -3.444]
  Call Extruder 0.01771
  MoveL (T14675) to (119.25, 111.86, 16.3) mm, rotated rx 180 ry 0 rz -180 deg; joints [2.298, 71.334, -37.656, 4.139, -33.747, -3.444]
  Call Extruder 0.08786
  MoveL (T14676) to (117.22, 109.83, 16.3) mm, rotated rx 180 ry 0 rz -180 deg; joints [2.298, 71.334, -37.656, 4.139, -33.747, -3.444]
  Call Extruder 0.01768
  MoveL (T14677) to (117.22, 110.41, 16.3) mm, rotated rx 180 ry 0 rz -180 deg; joints [2.298, 71.334, -37.656, 4.139, -33.747, -3.444]
  Call Extruder 0.08087
  MoveL (T14678) to (119.09, 112.28, 16.3) mm, rotated rx 180 ry 0 rz -180 deg; joints [2.359, 71.342, -37.67, 4.249, -33.744, -3.536]
  Set speed (45.0 mm/s)
  Call Extruder -1.6
  MoveL (T14679) to (119.09, 112.28, 16.3) mm, rotated rx 180 ry 0 rz -180 deg; joints [2.359, 71.342, -37.67, 4.249, -33.744, -3.536]
  Set speed (120.0 mm/s)
  MoveL (T14680) to (119.09, 112.28, 16.3) mm, rotated rx 180 ry 0 rz -180 deg; joints [1.42, 68.547, -32.412, 2.407, -36.159, -1.944]
  Call Extruder -0.38
  MoveL (T14681) to (118.34, 111.52, 16.3) mm, rotated rx 180 ry 0 rz -180 deg; joints [1.42, 68.547, -32.412, 2.407, -36.159, -1.944]
  Set speed (45.0 mm/s)
  Call Extruder -0.02
  MoveL (T14682) to (118.34, 111.52, 16.3) mm, rotated rx 180 ry 0 rz -180 deg; joints [1.42, 68.547, -32.412, 2.407, -36.159, -1.944]
  Set speed (150.0 mm/s)
  MoveL (T14683) to (118.34, 111.52, 18.3) mm, rotated rx 180 ry 0 rz -180 deg; joints [1.421, 68.386, -32.109, 2.401, -36.301, -1.936]
  MoveL (T14684) to (116.49, 107.94, 18.3) mm, rotated rx 180 ry 0 rz -180 deg; joints [1.421, 68.386, -32.109, 2.401, -36.301, -1.936]
  MoveL (T14685) to (116.49, 107.94, 16.3) mm, rotated rx 180 ry 0 rz -180 deg; joints [1.421, 68.386, -32.109, 2.401, -36.301, -1.936]
  Set speed (40.0 mm/s)
  Call Extruder 2.0
  MoveL (T14686) to (116.49, 107.94, 16.3) mm, rotated rx 180 ry 0 rz -180 deg; joints [1.421, 68.386, -32.109, 2.401, -36.301, -1.936]
  Call Extruder 0.17708
  MoveL (T14687) to (112.39, 103.84, 16.3) mm, rotated rx 180 ry 0 rz -180 deg; joints [2.42, 71.349, -37.685, 4.36, -33.741, -3.627]
  Call Extruder 0.01769
  MoveL (T14688) to (111.82, 103.84, 16.3) mm, rotated rx 180 ry 0 rz -180 deg; joints [2.42, 71.349, -37.685, 4.36, -33.741, -3.627]
  Call Extruder 0.16915
  MoveL (T14689) to (115.72, 107.75, 16.3) mm, rotated rx 180 ry 0 rz -180 deg; joints [2.481, 71.357, -37.699, 4.47, -33.738, -3.719]
  Call Extruder 0.01769
  MoveL (T14690) to (115.15, 107.75, 16.3) mm, rotated rx 180 ry 0 rz -180 deg; joints [2.481, 71.357, -37.699, 4.47, -33.738, -3.719]
  Call Extruder 0.16915
  MoveL (T14691) to (111.24, 103.84, 16.3) mm, rotated rx 180 ry 0 rz -180 deg; joints [2.481, 71.357, -37.699, 4.47, -33.738, -3.719]
  Call Extruder 0.01769
  MoveL (T14692) to (110.66, 103.84, 16.3) mm, rotated rx 180 ry 0 rz -180 deg; joints [1.423, 68.225, -31.808, 2.396, -36.442, -1.928]
  Call Extruder 0.16915
  MoveL (T14693) to (114.57, 107.75, 16.3) mm, rotated rx 180 ry 0 rz -180 deg; joints [1.423, 68.225, -31.808, 2.396, -36.442, -1.928]
  Call Extruder 0.01769
  MoveL (T14694) to (113.99, 107.75, 16.3) mm, rotated rx 180 ry 0 rz -180 deg; joints [1.424, 68.067, -31.509, 2.391, -36.582, -1.92]
  Call Extruder 0.16915
  MoveL (T14695) to (110.08, 103.84, 16.3) mm, rotated rx 180 ry 0 rz -180 deg; joints [1.424, 68.067, -31.509, 2.391, -36.582, -1.92]
  Call Extruder 0.01769
  MoveL (T14696) to (109.5, 103.84, 16.3) mm, rotated rx 180 ry 0 rz -180 deg; joints [1.424, 68.067, -31.509, 2.391, -36.582, -1.92]
  Call Extruder 0.11483
  MoveL (T14697) to (112.16, 106.5, 16.3) mm, rotated rx 180 ry 0 rz -180 deg; joints [2.542, 71.365, -37.714, 4.58, -33.735, -3.811]
  Call Extruder 0.01251
  MoveL (T14698) to (111.87, 106.79, 16.3) mm, rotated rx 180 ry 0 rz -180 deg; joints [2.542, 71.365, -37.714, 4.58, -33.735, -3.811]
  Call Extruder 0.12733
  MoveL (T14699) to (108.92, 103.84, 16.3) mm, rotated rx 180 ry 0 rz -180 deg; joints [2.603, 71.373, -37.73, 4.69, -33.732, -3.903]
  Call Extruder 0.01769
  MoveL (T14700) to (108.35, 103.84, 16.3) mm, rotated rx 180 ry 0 rz -180 deg; joints [2.603, 71.373, -37.73, 4.69, -33.732, -3.903]
  Call Extruder 0.13984
  MoveL (T14701) to (111.58, 107.08, 16.3) mm, rotated rx 180 ry 0 rz -180 deg; joints [1.426, 67.909, -31.212, 2.385, -36.721, -1.912]
  Call Extruder 0.01251
  MoveL (T14702) to (111.29, 107.36, 16.3) mm, rotated rx 180 ry 0 rz -180 deg; joints [1.428, 67.751, -30.916, 2.38, -36.859, -1.905]
  Call Extruder 0.15235
  MoveL (T14703) to (107.77, 103.84, 16.3) mm, rotated rx 180 ry 0 rz -180 deg; joints [1.428, 67.751, -30.916, 2.38, -36.859, -1.905]
  Call Extruder 0.01769
  MoveL (T14704) to (107.19, 103.84, 16.3) mm, rotated rx 180 ry 0 rz -180 deg; joints [2.663, 71.381, -37.746, 4.801, -33.729, -3.995]
  Call Extruder 0.16485
  MoveL (T14705) to (111, 107.65, 16.3) mm, rotated rx 180 ry 0 rz -180 deg; joints [2.663, 71.381, -37.746, 4.801, -33.729, -3.995]
  Call Extruder 0.00339
  MoveL (T14706) to (110.92, 107.73, 16.3) mm, rotated rx 180 ry 0 rz -180 deg; joints [2.663, 71.381, -37.746, 4.801, -33.729, -3.995]
  Call Extruder 0.00168
  MoveL (T14707) to (110.87, 107.75, 16.3) mm, rotated rx 180 ry 0 rz -180 deg; joints [2.663, 71.381, -37.746, 4.801, -33.729, -3.995]
  Call Extruder 0.0107
  MoveL (T14708) to (110.52, 107.75, 16.3) mm, rotated rx 180 ry 0 rz -180 deg; joints [2.724, 71.39, -37.762, 4.911, -33.726, -4.088]
  Call Extruder 0.16915
  MoveL (T14709) to (106.61, 103.84, 16.3) mm, rotated rx 180 ry 0 rz -180 deg; joints [2.724, 71.39, -37.762, 4.911, -33.726, -4.088]
  Call Extruder 0.01769
  MoveL (T14710) to (106.03, 103.84, 16.3) mm, rotated rx 180 ry 0 rz -180 deg; joints [1.429, 67.595, -30.622, 2.375, -36.997, -1.897]
  Call Extruder 0.16915
  MoveL (T14711) to (109.94, 107.75, 16.3) mm, rotated rx 180 ry 0 rz -180 deg; joints [1.429, 67.595, -30.622, 2.375, -36.997, -1.897]
  Call Extruder 0.01769
  MoveL (T14712) to (109.36, 107.75, 16.3) mm, rotated rx 180 ry 0 rz -180 deg; joints [1.431, 67.44, -30.33, 2.37, -37.133, -1.89]
  Call Extruder 0.16915
  MoveL (T14713) to (105.45, 103.84, 16.3) mm, rotated rx 180 ry 0 rz -180 deg; joints [1.431, 67.44, -30.33, 2.37, -37.133, -1.89]
  Call Extruder 0.01769
  MoveL (T14714) to (104.88, 103.84, 16.3) mm, rotated rx 180 ry 0 rz -180 deg; joints [2.785, 71.399, -37.778, 5.021, -33.722, -4.18]
  Call Extruder 0.16915
  MoveL (T14715) to (108.79, 107.75, 16.3) mm, rotated rx 180 ry 0 rz -180 deg; joints [2.785, 71.399, -37.778, 5.021, -33.722, -4.18]
  Call Extruder 0.01769
  MoveL (T14716) to (108.21, 107.75, 16.3) mm, rotated rx 180 ry 0 rz -180 deg; joints [2.785, 71.399, -37.778, 5.021, -33.722, -4.18]
  Call Extruder 0.16005
  MoveL (T14717) to (104.51, 104.06, 16.3) mm, rotated rx 180 ry 0 rz -180 deg; joints [2.785, 71.399, -37.778, 5.021, -33.722, -4.18]
  Call Extruder 0.01768
  MoveL (T14718) to (104.51, 104.63, 16.3) mm, rotated rx 180 ry 0 rz -180 deg; joints [2.846, 71.408, -37.795, 5.132, -33.719, -4.272]
  Call Extruder 0.13504
  MoveL (T14719) to (107.63, 107.75, 16.3) mm, rotated rx 180 ry 0 rz -180 deg; joints [2.846, 71.408, -37.795, 5.132, -33.719, -4.272]
  Call Extruder 0.01769
  MoveL (T14720) to (107.05, 107.75, 16.3) mm, rotated rx 180 ry 0 rz -180 deg; joints [1.432, 67.285, -30.04, 2.366, -37.269, -1.883]
  Call Extruder 0.11004
  MoveL (T14721) to (104.51, 105.21, 16.3) mm, rotated rx 180 ry 0 rz -180 deg; joints [1.432, 67.285, -30.04, 2.366, -37.269, -1.883]
  Call Extruder 0.01678
  MoveL (T14722) to (104.51, 105.76, 16.3) mm, rotated rx 180 ry 0 rz -180 deg; joints [1.432, 67.285, -30.04, 2.366, -37.269, -1.883]
  Call Extruder 0.00167
  MoveL (T14723) to (104.53, 105.81, 16.3) mm, rotated rx 180 ry 0 rz -180 deg; joints [1.434, 67.132, -29.751, 2.361, -37.405, -1.876]
  Call Extruder 0.09205
  MoveL (T14724) to (106.66, 107.94, 16.3) mm, rotated rx 180 ry 0 rz -180 deg; joints [1.434, 67.132, -29.751, 2.361, -37.405, -1.876]
  Set speed (45.0 mm/s)
  Call Extruder -1.6
  MoveL (T14725) to (106.66, 107.94, 16.3) mm, rotated rx 180 ry 0 rz -180 deg; joints [1.434, 67.132, -29.751, 2.361, -37.405, -1.876]
  Set speed (120.0 mm/s)
  MoveL (T14726) to (106.66, 107.94, 16.3) mm, rotated rx 180 ry 0 rz -180 deg; joints [2.907, 71.417, -37.812, 5.242, -33.715, -4.364]
  Call Extruder -0.38
  MoveL (T14727) to (105.9, 107.18, 16.3) mm, rotated rx 180 ry 0 rz -180 deg; joints [2.907, 71.417, -37.812, 5.242, -33.715, -4.364]
  Set speed (45.0 mm/s)
  Call Extruder -0.02
  MoveL (T14728) to (105.9, 107.18, 16.3) mm, rotated rx 180 ry 0 rz -180 deg; joints [2.907, 71.417, -37.812, 5.242, -33.715, -4.364]
  Set speed (150.0 mm/s)
  MoveL (T14729) to (105.9, 107.18, 18.3) mm, rotated rx 180 ry 0 rz -180 deg; joints [2.968, 71.426, -37.83, 5.353, -33.712, -4.457]
  MoveL (T14730) to (104.34, 103.54, 18.3) mm, rotated rx 180 ry 0 rz -180 deg; joints [2.968, 71.426, -37.83, 5.353, -33.712, -4.457]
  MoveL (T14731) to (104.34, 103.54, 16.5) mm, rotated rx 180 ry 0 rz -180 deg; joints [2.968, 71.426, -37.83, 5.353, -33.712, -4.457]
  Set speed (40.0 mm/s)
  Call Extruder 2.0
  MoveL (T14732) to (104.34, 103.54, 16.5) mm, rotated rx 180 ry 0 rz -180 deg; joints [1.435, 66.979, -29.464, 2.356, -37.539, -1.869]
  Set speed (36.8 mm/s)
  MoveL (T14733) to (104.34, 103.54, 16.5) mm, rotated rx 180 ry 0 rz -180 deg; joints [1.435, 66.979, -29.464, 2.356, -37.539, -1.869]
  Call Extruder 0.52159
  MoveL (T14734) to (121.46, 103.54, 16.5) mm, rotated rx 180 ry 0 rz -180 deg; joints [1.435, 66.979, -29.464, 2.356, -37.539, -1.869]
  Call Extruder 0.54596
  MoveL (T14735) to (121.46, 121.46, 16.5) mm, rotated rx 180 ry 0 rz -180 deg; joints [1.435, 66.979, -29.464, 2.356, -37.539, -1.869]
  Call Extruder 0.54596
  MoveL (T14736) to (103.54, 121.46, 16.5) mm, rotated rx 180 ry 0 rz -180 deg; joints [1.437, 66.827, -29.178, 2.352, -37.672, -1.862]
  Call Extruder 0.54596
  MoveL (T14737) to (103.54, 103.54, 16.5) mm, rotated rx 180 ry 0 rz -180 deg; joints [1.437, 66.827, -29.178, 2.352, -37.672, -1.862]
  Call Extruder 0.02254
  MoveL (T14738) to (104.28, 103.54, 16.5) mm, rotated rx 180 ry 0 rz -180 deg; joints [1.437, 66.827, -29.178, 2.352, -37.672, -1.862]
  Set speed (150.0 mm/s)
  MoveL (T14739) to (103.53, 103.13, 16.5) mm, rotated rx 180 ry 0 rz -180 deg; joints [3.029, 71.436, -37.848, 5.463, -33.708, -4.549]
  Set speed (36.8 mm/s)
  MoveL (T14740) to (103.53, 103.13, 16.5) mm, rotated rx 180 ry 0 rz -180 deg; joints [3.029, 71.436, -37.848, 5.463, -33.708, -4.549]
  Call Extruder 0.55858
  MoveL (T14741) to (121.87, 103.13, 16.5) mm, rotated rx 180 ry 0 rz -180 deg; joints [3.029, 71.436, -37.848, 5.463, -33.708, -4.549]
  Call Extruder 0.57077
  MoveL (T14742) to (121.87, 121.87, 16.5) mm, rotated rx 180 ry 0 rz -180 deg; joints [3.09, 71.446, -37.866, 5.574, -33.705, -4.641]
  Call Extruder 0.57077
  MoveL (T14743) to (103.13, 121.87, 16.5) mm, rotated rx 180 ry 0 rz -180 deg; joints [3.09, 71.446, -37.866, 5.574, -33.705, -4.641]
  Call Extruder 0.57077
  MoveL (T14744) to (103.13, 103.13, 16.5) mm, rotated rx 180 ry 0 rz -180 deg; joints [3.09, 71.446, -37.866, 5.574, -33.705, -4.641]
  Call Extruder 0.01036
  MoveL (T14745) to (103.47, 103.13, 16.5) mm, rotated rx 180 ry 0 rz -180 deg; joints [1.439, 66.677, -28.895, 2.347, -37.805, -1.855]
  Set speed (150.0 mm/s)
  MoveL (T14746) to (102.72, 102.81, 16.5) mm, rotated rx 180 ry 0 rz -180 deg; joints [1.439, 66.677, -28.895, 2.347, -37.805, -1.855]
  Set speed (25.0 mm/s)
  MoveL (T14747) to (102.72, 102.81, 16.5) mm, rotated rx 180 ry 0 rz -180 deg; joints [1.439, 66.677, -28.895, 2.347, -37.805, -1.855]
  Call Extruder 0.00259
  MoveL (T14748) to (102.72, 102.72, 16.5) mm, rotated rx 180 ry 0 rz -180 deg; joints [1.439, 66.677, -28.895, 2.347, -37.805, -1.855]
  Call Extruder 0.59557
  MoveL (T14749) to (122.28, 102.72, 16.5) mm, rotated rx 180 ry 0 rz -180 deg; joints [1.44, 66.526, -28.612, 2.343, -37.937, -1.848]
  Call Extruder 0.59557
  MoveL (T14750) to (122.28, 122.28, 16.5) mm, rotated rx 180 ry 0 rz -180 deg; joints [1.44, 66.526, -28.612, 2.343, -37.937, -1.848]
  Call Extruder 0.59557
  MoveL (T14751) to (102.72, 122.28, 16.5) mm, rotated rx 180 ry 0 rz -180 deg; joints [3.15, 71.456, -37.885, 5.684, -33.701, -4.734]
  Call Extruder 0.59115
  MoveL (T14752) to (102.72, 102.87, 16.5) mm, rotated rx 180 ry 0 rz -180 deg; joints [3.211, 71.466, -37.904, 5.795, -33.697, -4.826]
  Set speed (150.0 mm/s)
  MoveL (T14753) to (102.78, 102.75, 16.5) mm, rotated rx 180 ry 0 rz -180 deg; joints [3.211, 71.466, -37.904, 5.795, -33.697, -4.826]
  Set speed (45.0 mm/s)
  Call Extruder -1.6
  MoveL (T14754) to (102.78, 102.75, 16.5) mm, rotated rx 180 ry 0 rz -180 deg; joints [3.211, 71.466, -37.904, 5.795, -33.697, -4.826]
  Set speed (120.0 mm/s)
  MoveL (T14755) to (102.78, 102.75, 16.5) mm, rotated rx 180 ry 0 rz -180 deg; joints [1.442, 66.377, -28.332, 2.339, -38.069, -1.842]
  Call Extruder -0.05166
  MoveL (T14756) to (102.72, 102.72, 16.5) mm, rotated rx 180 ry 0 rz -180 deg; joints [1.442, 66.377, -28.332, 2.339, -38.069, -1.842]
  Call Extruder -0.32834
  MoveL (T14757) to (103.65, 102.72, 16.5) mm, rotated rx 180 ry 0 rz -180 deg; joints [1.505, 66.381, -28.339, 2.441, -38.067, -1.922]
  Set speed (45.0 mm/s)
  Call Extruder -0.02
  MoveL (T14758) to (103.65, 102.72, 16.5) mm, rotated rx 180 ry 0 rz -180 deg; joints [1.505, 66.381, -28.339, 2.441, -38.067, -1.922]
  Set speed (150.0 mm/s)
  MoveL (T14759) to (103.65, 102.72, 18.5) mm, rotated rx 180 ry 0 rz -180 deg; joints [3.215, 71.284, -37.561, 5.777, -33.857, -4.802]
  MoveL (T14760) to (103.84, 106.29, 18.5) mm, rotated rx 180 ry 0 rz -180 deg; joints [3.215, 71.284, -37.561, 5.777, -33.857, -4.802]
  MoveL (T14761) to (103.84, 106.29, 16.5) mm, rotated rx 180 ry 0 rz -180 deg; joints [3.218, 71.103, -37.221, 5.759, -34.016, -4.779]
  Set speed (40.0 mm/s)
  Call Extruder 2.0
  MoveL (T14762) to (103.84, 106.29, 16.5) mm, rotated rx 180 ry 0 rz -180 deg; joints [3.218, 71.103, -37.221, 5.759, -34.016, -4.779]
  Set speed (36.8 mm/s)
  MoveL (T14763) to (103.84, 106.29, 16.5) mm, rotated rx 180 ry 0 rz -180 deg; joints [1.568, 66.385, -28.346, 2.543, -38.066, -2.003]
  Call Extruder 0.07441
  MoveL (T14764) to (103.84, 103.84, 16.5) mm, rotated rx 180 ry 0 rz -180 deg; joints [1.568, 66.385, -28.346, 2.543, -38.066, -2.003]
  Call Extruder 0.0111
  MoveL (T14765) to (104.1, 104.1, 16.5) mm, rotated rx 180 ry 0 rz -180 deg; joints [1.568, 66.385, -28.346, 2.543, -38.066, -2.003]
  Call Extruder 0.05294
  MoveL (T14766) to (104.1, 105.84, 16.5) mm, rotated rx 180 ry 0 rz -180 deg; joints [1.631, 66.389, -28.354, 2.645, -38.065, -2.083]
  Call Extruder 0.00661
  MoveL (T14767) to (104.18, 106.04, 16.5) mm, rotated rx 180 ry 0 rz -180 deg; joints [1.631, 66.389, -28.354, 2.645, -38.065, -2.083]
  Call Extruder 0.02065
  MoveL (T14768) to (104.66, 106.52, 16.5) mm, rotated rx 180 ry 0 rz -180 deg; joints [3.222, 70.924, -36.884, 5.742, -34.173, -4.756]
  Call Extruder 0.03528
  MoveL (T14769) to (103.84, 107.34, 16.5) mm, rotated rx 180 ry 0 rz -180 deg; joints [3.222, 70.924, -36.884, 5.742, -34.173, -4.756]
  Call Extruder 0.03385
  MoveL (T14770) to (103.84, 108.45, 16.5) mm, rotated rx 180 ry 0 rz -180 deg; joints [3.222, 70.924, -36.884, 5.742, -34.173, -4.756]
  Call Extruder 0.54738
  MoveL (T14771) to (116.55, 121.16, 16.5) mm, rotated rx 180 ry 0 rz -180 deg; joints [3.225, 70.746, -36.549, 5.725, -34.33, -4.733]
  Call Extruder 0.03385
  MoveL (T14772) to (117.66, 121.16, 16.5) mm, rotated rx 180 ry 0 rz -180 deg; joints [1.694, 66.393, -28.362, 2.748, -38.063, -2.164]
  Call Extruder 0.0423
  MoveL (T14773) to (118.64, 120.17, 16.5) mm, rotated rx 180 ry 0 rz -180 deg; joints [1.694, 66.393, -28.362, 2.748, -38.063, -2.164]
  Call Extruder 0.01225
  MoveL (T14774) to (118.93, 120.46, 16.5) mm, rotated rx 180 ry 0 rz -180 deg; joints [1.694, 66.393, -28.362, 2.748, -38.063, -2.164]
  Call Extruder 0.00661
  MoveL (T14775) to (119.13, 120.54, 16.5) mm, rotated rx 180 ry 0 rz -180 deg; joints [1.757, 66.398, -28.371, 2.85, -38.062, -2.245]
  Call Extruder 0.04314
  MoveL (T14776) to (120.54, 120.54, 16.5) mm, rotated rx 180 ry 0 rz -180 deg; joints [1.757, 66.398, -28.371, 2.85, -38.062, -2.245]
  Call Extruder 0.02637
  MoveL (T14777) to (121.16, 121.16, 16.5) mm, rotated rx 180 ry 0 rz -180 deg; joints [1.757, 66.398, -28.371, 2.85, -38.062, -2.245]
  Call Extruder 0.07441
  MoveL (T14778) to (118.71, 121.16, 16.5) mm, rotated rx 180 ry 0 rz -180 deg; joints [3.228, 70.569, -36.217, 5.708, -34.485, -4.71]
  Set speed (45.0 mm/s)
  Call Extruder -1.6
  MoveL (T14779) to (118.71, 121.16, 16.5) mm, rotated rx 180 ry 0 rz -180 deg; joints [3.228, 70.569, -36.217, 5.708, -34.485, -4.71]
  Set speed (120.0 mm/s)
  MoveL (T14780) to (118.71, 121.16, 16.5) mm, rotated rx 180 ry 0 rz -180 deg; joints [3.228, 70.569, -36.217, 5.708, -34.485, -4.71]
  Call Extruder -0.38
  MoveL (T14781) to (119.78, 121.16, 16.5) mm, rotated rx 180 ry 0 rz -180 deg; joints [3.232, 70.394, -35.888, 5.692, -34.639, -4.688]
  Set speed (45.0 mm/s)
  Call Extruder -0.02
  MoveL (T14782) to (119.78, 121.16, 16.5) mm, rotated rx 180 ry 0 rz -180 deg; joints [3.232, 70.394, -35.888, 5.692, -34.639, -4.688]
  Set speed (150.0 mm/s)
  MoveL (T14783) to (119.78, 121.16, 18.5) mm, rotated rx 180 ry 0 rz -180 deg; joints [1.82, 66.403, -28.379, 2.952, -38.06, -2.325]
  MoveL (T14784) to (121.34, 119.42, 18.5) mm, rotated rx 180 ry 0 rz -180 deg; joints [1.82, 66.403, -28.379, 2.952, -38.06, -2.325]
  MoveL (T14785) to (121.34, 119.42, 16.5) mm, rotated rx 180 ry 0 rz -180 deg; joints [1.882, 66.407, -28.388, 3.055, -38.059, -2.406]
  Set speed (40.0 mm/s)
  Call Extruder 2.0
  MoveL (T14786) to (121.34, 119.42, 16.5) mm, rotated rx 180 ry 0 rz -180 deg; joints [1.882, 66.407, -28.388, 3.055, -38.059, -2.406]
  Set speed (36.8 mm/s)
  MoveL (T14787) to (121.34, 119.42, 16.5) mm, rotated rx 180 ry 0 rz -180 deg; joints [3.235, 70.22, -35.561, 5.676, -34.791, -4.667]
  Call Extruder 0.03108
  MoveL (T14788) to (120.62, 120.14, 16.5) mm, rotated rx 180 ry 0 rz -180 deg; joints [3.235, 70.22, -35.561, 5.676, -34.791, -4.667]
  Call Extruder 0.01774
  MoveL (T14789) to (120.04, 120.14, 16.5) mm, rotated rx 180 ry 0 rz -180 deg; joints [3.239, 70.048, -35.237, 5.661, -34.943, -4.645]
  Call Extruder 0.04823
  MoveL (T14790) to (121.16, 119.02, 16.5) mm, rotated rx 180 ry 0 rz -180 deg; joints [3.239, 70.048, -35.237, 5.661, -34.943, -4.645]
  Call Extruder 0.01777
  MoveL (T14791) to (121.16, 118.44, 16.5) mm, rotated rx 180 ry 0 rz -180 deg; joints [3.239, 70.048, -35.237, 5.661, -34.943, -4.645]
  Call Extruder 0.07333
  MoveL (T14792) to (119.47, 120.14, 16.5) mm, rotated rx 180 ry 0 rz -180 deg; joints [1.945, 66.412, -28.398, 3.157, -38.057, -2.487]
  Call Extruder 0.00784
  MoveL (T14793) to (119.21, 120.14, 16.5) mm, rotated rx 180 ry 0 rz -180 deg; joints [1.945, 66.412, -28.398, 3.157, -38.057, -2.487]
  Call Extruder 0.00169
  MoveL (T14794) to (119.16, 120.11, 16.5) mm, rotated rx 180 ry 0 rz -180 deg; joints [1.945, 66.412, -28.398, 3.157, -38.057, -2.487]
  Call Extruder 0.00545
  MoveL (T14795) to (119.03, 119.99, 16.5) mm, rotated rx 180 ry 0 rz -180 deg; joints [1.945, 66.412, -28.398, 3.157, -38.057, -2.487]
  Call Extruder 0.09207
  MoveL (T14796) to (121.16, 117.86, 16.5) mm, rotated rx 180 ry 0 rz -180 deg; joints [2.008, 66.418, -28.408, 3.259, -38.055, -2.567]
  Call Extruder 0.01777
  MoveL (T14797) to (121.16, 117.28, 16.5) mm, rotated rx 180 ry 0 rz -180 deg; joints [3.242, 69.877, -34.914, 5.646, -35.093, -4.624]
  Call Extruder 0.10462
  MoveL (T14798) to (118.74, 119.7, 16.5) mm, rotated rx 180 ry 0 rz -180 deg; joints [3.242, 69.877, -34.914, 5.646, -35.093, -4.624]
  Call Extruder 0.01256
  MoveL (T14799) to (118.45, 119.41, 16.5) mm, rotated rx 180 ry 0 rz -180 deg; joints [3.246, 69.707, -34.595, 5.631, -35.243, -4.604]
  Call Extruder 0.11718
  MoveL (T14800) to (121.16, 116.7, 16.5) mm, rotated rx 180 ry 0 rz -180 deg; joints [3.246, 69.707, -34.595, 5.631, -35.243, -4.604]
  Call Extruder 0.01777
  MoveL (T14801) to (121.16, 116.13, 16.5) mm, rotated rx 180 ry 0 rz -180 deg; joints [2.071, 66.423, -28.417, 3.362, -38.053, -2.648]
  Call Extruder 0.12973
  MoveL (T14802) to (118.16, 119.12, 16.5) mm, rotated rx 180 ry 0 rz -180 deg; joints [2.134, 66.428, -28.428, 3.464, -38.051, -2.729]
  Call Extruder 0.01256
  MoveL (T14803) to (117.87, 118.83, 16.5) mm, rotated rx 180 ry 0 rz -180 deg; joints [2.134, 66.428, -28.428, 3.464, -38.051, -2.729]
  Call Extruder 0.14228
  MoveL (T14804) to (121.16, 115.55, 16.5) mm, rotated rx 180 ry 0 rz -180 deg; joints [3.249, 69.538, -34.277, 5.616, -35.391, -4.583]
  Call Extruder 0.01777
  MoveL (T14805) to (121.16, 114.97, 16.5) mm, rotated rx 180 ry 0 rz -180 deg; joints [3.253, 69.371, -33.962, 5.602, -35.538, -4.563]
  Call Extruder 0.15484
  MoveL (T14806) to (117.58, 118.54, 16.5) mm, rotated rx 180 ry 0 rz -180 deg; joints [3.253, 69.371, -33.962, 5.602, -35.538, -4.563]
  Call Extruder 0.01256
  MoveL (T14807) to (117.3, 118.25, 16.5) mm, rotated rx 180 ry 0 rz -180 deg; joints [2.197, 66.434, -28.438, 3.566, -38.049, -2.81]
  Call Extruder 0.16739
  MoveL (T14808) to (121.16, 114.39, 16.5) mm, rotated rx 180 ry 0 rz -180 deg; joints [2.197, 66.434, -28.438, 3.566, -38.049, -2.81]
  Call Extruder 0.01777
  MoveL (T14809) to (121.16, 113.81, 16.5) mm, rotated rx 180 ry 0 rz -180 deg; joints [2.197, 66.434, -28.438, 3.566, -38.049, -2.81]
  Call Extruder 0.17073
  MoveL (T14810) to (117.22, 117.75, 16.5) mm, rotated rx 180 ry 0 rz -180 deg; joints [2.26, 66.44, -28.449, 3.669, -38.048, -2.891]
  Call Extruder 0.01778
  MoveL (T14811) to (117.22, 117.17, 16.5) mm, rotated rx 180 ry 0 rz -180 deg; joints [2.26, 66.44, -28.449, 3.669, -38.048, -2.891]
  Call Extruder 0.17072
  MoveL (T14812) to (121.16, 113.23, 16.5) mm, rotated rx 180 ry 0 rz -180 deg; joints [2.26, 66.44, -28.449, 3.669, -38.048, -2.891]
  Call Extruder 0.01777
  MoveL (T14813) to (121.16, 112.65, 16.5) mm, rotated rx 180 ry 0 rz -180 deg; joints [3.256, 69.204, -33.649, 5.588, -35.684, -4.544]
  Call Extruder 0.17071
  MoveL (T14814) to (117.22, 116.59, 16.5) mm, rotated rx 180 ry 0 rz -180 deg; joints [3.256, 69.204, -33.649, 5.588, -35.684, -4.544]
  Call Extruder 0.01778
  MoveL (T14815) to (117.22, 116.01, 16.5) mm, rotated rx 180 ry 0 rz -180 deg; joints [3.256, 69.204, -33.649, 5.588, -35.684, -4.544]
  Call Extruder 0.17069
  MoveL (T14816) to (121.16, 112.07, 16.5) mm, rotated rx 180 ry 0 rz -180 deg; joints [3.26, 69.039, -33.339, 5.574, -35.829, -4.524]
  Call Extruder 0.01777
  MoveL (T14817) to (121.16, 111.49, 16.5) mm, rotated rx 180 ry 0 rz -180 deg; joints [3.26, 69.039, -33.339, 5.574, -35.829, -4.524]
  Call Extruder 0.17068
  MoveL (T14818) to (117.22, 115.43, 16.5) mm, rotated rx 180 ry 0 rz -180 deg; joints [2.323, 66.446, -28.461, 3.771, -38.046, -2.971]
  Call Extruder 0.01778
  MoveL (T14819) to (117.22, 114.85, 16.5) mm, rotated rx 180 ry 0 rz -180 deg; joints [2.323, 66.446, -28.461, 3.771, -38.046, -2.971]
  Call Extruder 0.17067
  MoveL (T14820) to (121.16, 110.91, 16.5) mm, rotated rx 180 ry 0 rz -180 deg; joints [2.386, 66.452, -28.472, 3.873, -38.043, -3.052]
  Call Extruder 0.01777
  MoveL (T14821) to (121.16, 110.33, 16.5) mm, rotated rx 180 ry 0 rz -180 deg; joints [2.386, 66.452, -28.472, 3.873, -38.043, -3.052]
  Call Extruder 0.17066
  MoveL (T14822) to (117.22, 114.27, 16.5) mm, rotated rx 180 ry 0 rz -180 deg; joints [2.386, 66.452, -28.472, 3.873, -38.043, -3.052]
  Call Extruder 0.01813
  MoveL (T14823) to (117.23, 113.68, 16.5) mm, rotated rx 180 ry 0 rz -180 deg; joints [3.263, 68.875, -33.03, 5.561, -35.974, -4.505]
  Call Extruder 0.17015
  MoveL (T14824) to (121.16, 109.75, 16.5) mm, rotated rx 180 ry 0 rz -180 deg; joints [3.263, 68.875, -33.03, 5.561, -35.974, -4.505]
  Call Extruder 0.01777
  MoveL (T14825) to (121.16, 109.17, 16.5) mm, rotated rx 180 ry 0 rz -180 deg; joints [3.263, 68.875, -33.03, 5.561, -35.974, -4.505]
  Call Extruder 0.11319
  MoveL (T14826) to (118.55, 111.78, 16.5) mm, rotated rx 180 ry 0 rz -180 deg; joints [3.263, 68.875, -33.03, 5.561, -35.974, -4.505]
  Call Extruder 0.01256
  MoveL (T14827) to (118.26, 111.49, 16.5) mm, rotated rx 180 ry 0 rz -180 deg; joints [3.267, 68.712, -32.723, 5.548, -36.117, -4.487]
  Call Extruder 0.12575
  MoveL (T14828) to (121.16, 108.59, 16.5) mm, rotated rx 180 ry 0 rz -180 deg; joints [3.267, 68.712, -32.723, 5.548, -36.117, -4.487]
  Call Extruder 0.01777
  MoveL (T14829) to (121.16, 108.01, 16.5) mm, rotated rx 180 ry 0 rz -180 deg; joints [2.449, 66.458, -28.484, 3.976, -38.041, -3.133]
  Call Extruder 0.13832
  MoveL (T14830) to (117.97, 111.2, 16.5) mm, rotated rx 180 ry 0 rz -180 deg; joints [2.449, 66.458, -28.484, 3.976, -38.041, -3.133]
  Call Extruder 0.01256
  MoveL (T14831) to (117.68, 110.91, 16.5) mm, rotated rx 180 ry 0 rz -180 deg; joints [2.449, 66.458, -28.484, 3.976, -38.041, -3.133]
  Call Extruder 0.15088
  MoveL (T14832) to (121.16, 107.43, 16.5) mm, rotated rx 180 ry 0 rz -180 deg; joints [2.512, 66.465, -28.496, 4.078, -38.039, -3.214]
  Call Extruder 0.01777
  MoveL (T14833) to (121.16, 106.86, 16.5) mm, rotated rx 180 ry 0 rz -180 deg; joints [2.512, 66.465, -28.496, 4.078, -38.039, -3.214]
  Call Extruder 0.16345
  MoveL (T14834) to (117.39, 110.62, 16.5) mm, rotated rx 180 ry 0 rz -180 deg; joints [3.27, 68.55, -32.418, 5.535, -36.259, -4.468]
  Call Extruder 0.00624
  MoveL (T14835) to (117.24, 110.48, 16.5) mm, rotated rx 180 ry 0 rz -180 deg; joints [3.27, 68.55, -32.418, 5.535, -36.259, -4.468]
  Call Extruder 0.00169
  MoveL (T14836) to (117.22, 110.43, 16.5) mm, rotated rx 180 ry 0 rz -180 deg; joints [3.27, 68.55, -32.418, 5.535, -36.259, -4.468]
  Call Extruder 0.00674
  MoveL (T14837) to (117.22, 110.21, 16.5) mm, rotated rx 180 ry 0 rz -180 deg; joints [3.274, 68.389, -32.116, 5.522, -36.401, -4.45]
  Call Extruder 0.1706
  MoveL (T14838) to (121.16, 106.28, 16.5) mm, rotated rx 180 ry 0 rz -180 deg; joints [3.274, 68.389, -32.116, 5.522, -36.401, -4.45]
  Call Extruder 0.01777
  MoveL (T14839) to (121.16, 105.7, 16.5) mm, rotated rx 180 ry 0 rz -180 deg; joints [3.274, 68.389, -32.116, 5.522, -36.401, -4.45]
  Call Extruder 0.17058
  MoveL (T14840) to (117.22, 109.63, 16.5) mm, rotated rx 180 ry 0 rz -180 deg; joints [2.575, 66.471, -28.509, 4.181, -38.037, -3.295]
  Call Extruder 0.01778
  MoveL (T14841) to (117.22, 109.05, 16.5) mm, rotated rx 180 ry 0 rz -180 deg; joints [2.575, 66.471, -28.509, 4.181, -38.037, -3.295]
  Call Extruder 0.17057
  MoveL (T14842) to (121.16, 105.12, 16.5) mm, rotated rx 180 ry 0 rz -180 deg; joints [2.575, 66.471, -28.509, 4.181, -38.037, -3.295]
  Call Extruder 0.01777
  MoveL (T14843) to (121.16, 104.54, 16.5) mm, rotated rx 180 ry 0 rz -180 deg; joints [2.638, 66.478, -28.521, 4.283, -38.035, -3.376]
  Call Extruder 0.17056
  MoveL (T14844) to (117.22, 108.47, 16.5) mm, rotated rx 180 ry 0 rz -180 deg; joints [2.638, 66.478, -28.521, 4.283, -38.035, -3.376]
  Call Extruder 0.01778
  MoveL (T14845) to (117.22, 107.89, 16.5) mm, rotated rx 180 ry 0 rz -180 deg; joints [3.277, 68.229, -31.815, 5.51, -36.541, -4.432]
  Call Extruder 0.16962
  MoveL (T14846) to (121.13, 103.98, 16.5) mm, rotated rx 180 ry 0 rz -180 deg; joints [3.277, 68.229, -31.815, 5.51, -36.541, -4.432]
  Call Extruder 0.01778
  MoveL (T14847) to (120.55, 103.98, 16.5) mm, rotated rx 180 ry 0 rz -180 deg; joints [3.281, 68.07, -31.516, 5.498, -36.681, -4.414]
  Call Extruder 0.16368
  MoveL (T14848) to (116.78, 107.75, 16.5) mm, rotated rx 180 ry 0 rz -180 deg; joints [3.281, 68.07, -31.516, 5.498, -36.681, -4.414]
  Call Extruder 0.01777
  MoveL (T14849) to (116.2, 107.75, 16.5) mm, rotated rx 180 ry 0 rz -180 deg; joints [2.7, 66.485, -28.534, 4.386, -38.032, -3.457]
  Call Extruder 0.16367
  MoveL (T14850) to (119.97, 103.98, 16.5) mm, rotated rx 180 ry 0 rz -180 deg; joints [2.7, 66.485, -28.534, 4.386, -38.032, -3.457]
  Call Extruder 0.00371
  MoveL (T14851) to (119.85, 103.98, 16.5) mm, rotated rx 180 ry 0 rz -180 deg; joints [2.7, 66.485, -28.534, 4.386, -38.032, -3.457]
  Call Extruder 0.00414
  MoveL (T14852) to (119.85, 103.84, 16.5) mm, rotated rx 180 ry 0 rz -180 deg; joints [2.763, 66.492, -28.548, 4.488, -38.03, -3.538]
  Call Extruder 0.00992
  MoveL (T14853) to (119.53, 103.84, 16.5) mm, rotated rx 180 ry 0 rz -180 deg; joints [2.763, 66.492, -28.548, 4.488, -38.03, -3.538]
  Call Extruder 0.16952
  MoveL (T14854) to (115.62, 107.75, 16.5) mm, rotated rx 180 ry 0 rz -180 deg; joints [3.285, 67.912, -31.219, 5.486, -36.82, -4.397]
  Call Extruder 0.01777
  MoveL (T14855) to (115.04, 107.75, 16.5) mm, rotated rx 180 ry 0 rz -180 deg; joints [3.285, 67.912, -31.219, 5.486, -36.82, -4.397]
  Call Extruder 0.16952
  MoveL (T14856) to (118.95, 103.84, 16.5) mm, rotated rx 180 ry 0 rz -180 deg; joints [3.285, 67.912, -31.219, 5.486, -36.82, -4.397]
  Call Extruder 0.01777
  MoveL (T14857) to (118.37, 103.84, 16.5) mm, rotated rx 180 ry 0 rz -180 deg; joints [3.288, 67.755, -30.923, 5.474, -36.958, -4.379]
  Call Extruder 0.16952
  MoveL (T14858) to (114.46, 107.75, 16.5) mm, rotated rx 180 ry 0 rz -180 deg; joints [3.288, 67.755, -30.923, 5.474, -36.958, -4.379]
  Call Extruder 0.01777
  MoveL (T14859) to (113.88, 107.75, 16.5) mm, rotated rx 180 ry 0 rz -180 deg; joints [3.288, 67.755, -30.923, 5.474, -36.958, -4.379]
  Call Extruder 0.16952
  MoveL (T14860) to (117.79, 103.84, 16.5) mm, rotated rx 180 ry 0 rz -180 deg; joints [2.826, 66.499, -28.562, 4.591, -38.027, -3.619]
  Call Extruder 0.01777
  MoveL (T14861) to (117.21, 103.84, 16.5) mm, rotated rx 180 ry 0 rz -180 deg; joints [2.826, 66.499, -28.562, 4.591, -38.027, -3.619]
  Call Extruder 0.16599
  MoveL (T14862) to (113.38, 107.67, 16.5) mm, rotated rx 180 ry 0 rz -180 deg; joints [2.826, 66.499, -28.562, 4.591, -38.027, -3.619]
  Call Extruder 0.01256
  MoveL (T14863) to (113.09, 107.38, 16.5) mm, rotated rx 180 ry 0 rz -180 deg; joints [2.889, 66.507, -28.576, 4.693, -38.025, -3.7]
  Call Extruder 0.15343
  MoveL (T14864) to (116.63, 103.84, 16.5) mm, rotated rx 180 ry 0 rz -180 deg; joints [2.889, 66.507, -28.576, 4.693, -38.025, -3.7]
  Call Extruder 0.01777
  MoveL (T14865) to (116.05, 103.84, 16.5) mm, rotated rx 180 ry 0 rz -180 deg; joints [3.292, 67.599, -30.63, 5.463, -37.095, -4.362]
  Call Extruder 0.14087
  MoveL (T14866) to (112.81, 107.09, 16.5) mm, rotated rx 180 ry 0 rz -180 deg; joints [3.292, 67.599, -30.63, 5.463, -37.095, -4.362]
  Call Extruder 0.01256
  MoveL (T14867) to (112.52, 106.8, 16.5) mm, rotated rx 180 ry 0 rz -180 deg; joints [3.295, 67.444, -30.338, 5.452, -37.231, -4.345]
  Call Extruder 0.12831
  MoveL (T14868) to (115.47, 103.84, 16.5) mm, rotated rx 180 ry 0 rz -180 deg; joints [3.295, 67.444, -30.338, 5.452, -37.231, -4.345]
  Call Extruder 0.01777
  MoveL (T14869) to (114.89, 103.84, 16.5) mm, rotated rx 180 ry 0 rz -180 deg; joints [3.295, 67.444, -30.338, 5.452, -37.231, -4.345]
  Call Extruder 0.11574
  MoveL (T14870) to (112.22, 106.51, 16.5) mm, rotated rx 180 ry 0 rz -180 deg; joints [2.952, 66.515, -28.59, 4.796, -38.022, -3.781]
  Call Extruder 0.00182
  MoveL (T14871) to (112.18, 106.47, 16.5) mm, rotated rx 180 ry 0 rz -180 deg; joints [2.952, 66.515, -28.59, 4.796, -38.022, -3.781]
  Call Extruder 0.05469
  MoveL (T14872) to (110.92, 107.73, 16.5) mm, rotated rx 180 ry 0 rz -180 deg; joints [3.015, 66.522, -28.605, 4.898, -38.019, -3.862]
  Call Extruder 0.00169
  MoveL (T14873) to (110.87, 107.75, 16.5) mm, rotated rx 180 ry 0 rz -180 deg; joints [3.015, 66.522, -28.605, 4.898, -38.019, -3.862]
  Call Extruder 0.01426
  MoveL (T14874) to (110.41, 107.75, 16.5) mm, rotated rx 180 ry 0 rz -180 deg; joints [3.015, 66.522, -28.605, 4.898, -38.019, -3.862]
  Call Extruder 0.16952
  MoveL (T14875) to (114.31, 103.84, 16.5) mm, rotated rx 180 ry 0 rz -180 deg; joints [3.299, 67.29, -30.048, 5.441, -37.367, -4.329]
  Call Extruder 0.01777
  MoveL (T14876) to (113.73, 103.84, 16.5) mm, rotated rx 180 ry 0 rz -180 deg; joints [3.299, 67.29, -30.048, 5.441, -37.367, -4.329]
  Call Extruder 0.16952
  MoveL (T14877) to (109.83, 107.75, 16.5) mm, rotated rx 180 ry 0 rz -180 deg; joints [3.299, 67.29, -30.048, 5.441, -37.367, -4.329]
  Call Extruder 0.01777
  MoveL (T14878) to (109.25, 107.75, 16.5) mm, rotated rx 180 ry 0 rz -180 deg; joints [3.302, 67.137, -29.76, 5.43, -37.501, -4.313]
  Call Extruder 0.16952
  MoveL (T14879) to (113.16, 103.84, 16.5) mm, rotated rx 180 ry 0 rz -180 deg; joints [3.302, 67.137, -29.76, 5.43, -37.501, -4.313]
  Call Extruder 0.01777
  MoveL (T14880) to (112.58, 103.84, 16.5) mm, rotated rx 180 ry 0 rz -180 deg; joints [3.077, 66.53, -28.619, 5.001, -38.017, -3.944]
  Call Extruder 0.16952
  MoveL (T14881) to (108.67, 107.75, 16.5) mm, rotated rx 180 ry 0 rz -180 deg; joints [3.14, 66.538, -28.635, 5.103, -38.014, -4.025]
  Call Extruder 0.01777
  MoveL (T14882) to (108.09, 107.75, 16.5) mm, rotated rx 180 ry 0 rz -180 deg; joints [3.14, 66.538, -28.635, 5.103, -38.014, -4.025]
  Call Extruder 0.16952
  MoveL (T14883) to (112, 103.84, 16.5) mm, rotated rx 180 ry 0 rz -180 deg; joints [3.14, 66.538, -28.635, 5.103, -38.014, -4.025]
  Call Extruder 0.01777
  MoveL (T14884) to (111.42, 103.84, 16.5) mm, rotated rx 180 ry 0 rz -180 deg; joints [3.14, 66.538, -28.635, 5.103, -38.014, -4.025]
  Call Extruder 0.16952
  MoveL (T14885) to (107.51, 107.75, 16.5) mm, rotated rx 180 ry 0 rz -180 deg; joints [3.306, 66.984, -29.474, 5.419, -37.635, -4.296]
  Call Extruder 0.01777
  MoveL (T14886) to (106.93, 107.75, 16.5) mm, rotated rx 180 ry 0 rz -180 deg; joints [3.31, 66.833, -29.188, 5.409, -37.768, -4.281]
  Call Extruder 0.16952
  MoveL (T14887) to (110.84, 103.84, 16.5) mm, rotated rx 180 ry 0 rz -180 deg; joints [3.31, 66.833, -29.188, 5.409, -37.768, -4.281]
  Call Extruder 0.01777
  MoveL (T14888) to (110.26, 103.84, 16.5) mm, rotated rx 180 ry 0 rz -180 deg; joints [3.203, 66.547, -28.65, 5.206, -38.011, -4.106]
  Call Extruder 0.16685
  MoveL (T14889) to (106.41, 107.69, 16.5) mm, rotated rx 180 ry 0 rz -180 deg; joints [3.203, 66.547, -28.65, 5.206, -38.011, -4.106]
  Call Extruder 0.01256
  MoveL (T14890) to (106.12, 107.4, 16.5) mm, rotated rx 180 ry 0 rz -180 deg; joints [3.203, 66.547, -28.65, 5.206, -38.011, -4.106]
  Call Extruder 0.15429
  MoveL (T14891) to (109.68, 103.84, 16.5) mm, rotated rx 180 ry 0 rz -180 deg; joints [3.266, 66.555, -28.666, 5.309, -38.008, -4.187]
  Call Extruder 0.01777
  MoveL (T14892) to (109.1, 103.84, 16.5) mm, rotated rx 180 ry 0 rz -180 deg; joints [3.266, 66.555, -28.666, 5.309, -38.008, -4.187]
  Call Extruder 0.14172
  MoveL (T14893) to (105.83, 107.11, 16.5) mm, rotated rx 180 ry 0 rz -180 deg; joints [3.332, 66.732, -28.999, 5.434, -37.858, -4.295]
  Call Extruder 0.01256
  MoveL (T14894) to (105.54, 106.82, 16.5) mm, rotated rx 180 ry 0 rz -180 deg; joints [3.332, 66.732, -28.999, 5.434, -37.858, -4.295]
  Call Extruder 0.12915
  MoveL (T14895) to (108.52, 103.84, 16.5) mm, rotated rx 180 ry 0 rz -180 deg; joints [3.332, 66.732, -28.999, 5.434, -37.858, -4.295]
  Call Extruder 0.01777
  MoveL (T14896) to (107.94, 103.84, 16.5) mm, rotated rx 180 ry 0 rz -180 deg; joints [3.332, 66.732, -28.999, 5.434, -37.858, -4.295]
  Call Extruder 0.11659
  MoveL (T14897) to (105.25, 106.53, 16.5) mm, rotated rx 180 ry 0 rz -180 deg; joints [3.332, 66.732, -28.999, 5.434, -37.858, -4.295]
  Call Extruder 0.01256
  MoveL (T14898) to (104.96, 106.24, 16.5) mm, rotated rx 180 ry 0 rz -180 deg; joints [3.332, 66.732, -28.999, 5.434, -37.858, -4.295]
  Call Extruder 0.10402
  MoveL (T14899) to (107.36, 103.84, 16.5) mm, rotated rx 180 ry 0 rz -180 deg; joints [3.332, 66.732, -28.999, 5.434, -37.858, -4.295]
  Call Extruder 0.01777
  MoveL (T14900) to (106.78, 103.84, 16.5) mm, rotated rx 180 ry 0 rz -180 deg; joints [3.332, 66.732, -28.999, 5.434, -37.858, -4.295]
  Call Extruder 0.09145
  MoveL (T14901) to (104.67, 105.95, 16.5) mm, rotated rx 180 ry 0 rz -180 deg; joints [3.332, 66.732, -28.999, 5.434, -37.858, -4.295]
  Call Extruder 0.00622
  MoveL (T14902) to (104.53, 105.81, 16.5) mm, rotated rx 180 ry 0 rz -180 deg; joints [3.332, 66.732, -28.999, 5.434, -37.858, -4.295]
  Call Extruder 0.00169
  MoveL (T14903) to (104.51, 105.76, 16.5) mm, rotated rx 180 ry 0 rz -180 deg; joints [3.332, 66.732, -28.999, 5.434, -37.858, -4.295]
  Call Extruder 0.00677
  MoveL (T14904) to (104.51, 105.54, 16.5) mm, rotated rx 180 ry 0 rz -180 deg; joints [3.332, 66.732, -28.999, 5.434, -37.858, -4.295]
  Call Extruder 0.07345
  MoveL (T14905) to (106.2, 103.84, 16.5) mm, rotated rx 180 ry 0 rz -180 deg; joints [3.332, 66.732, -28.999, 5.434, -37.858, -4.295]
  Call Extruder 0.01777
  MoveL (T14906) to (105.62, 103.84, 16.5) mm, rotated rx 180 ry 0 rz -180 deg; joints [3.332, 66.732, -28.999, 5.434, -37.858, -4.295]
  Call Extruder 0.04831
  MoveL (T14907) to (104.51, 104.96, 16.5) mm, rotated rx 180 ry 0 rz -180 deg; joints [3.266, 66.555, -28.666, 5.309, -38.008, -4.187]
  Call Extruder 0.01778
  MoveL (T14908) to (104.51, 104.38, 16.5) mm, rotated rx 180 ry 0 rz -180 deg; joints [3.25, 66.553, -28.662, 5.282, -38.009, -4.166]
  Call Extruder 0.03112
  MoveL (T14909) to (105.23, 103.66, 16.5) mm, rotated rx 180 ry 0 rz -180 deg; joints [3.25, 66.553, -28.662, 5.282, -38.009, -4.166]
  Set speed (45.0 mm/s)
  Call Extruder -1.6
  MoveL (T14910) to (105.23, 103.66, 16.5) mm, rotated rx 180 ry 0 rz -180 deg; joints [3.25, 66.553, -28.662, 5.282, -38.009, -4.166]
  Set speed (120.0 mm/s)
  MoveL (T14911) to (105.23, 103.66, 16.5) mm, rotated rx 180 ry 0 rz -180 deg; joints [3.25, 66.553, -28.662, 5.282, -38.009, -4.166]
  Call Extruder -0.36151
  MoveL (T14912) to (104.51, 104.38, 16.5) mm, rotated rx 180 ry 0 rz -180 deg; joints [3.25, 66.553, -28.662, 5.282, -38.009, -4.166]
  Call Extruder -0.01849
  MoveL (T14913) to (104.51, 104.43, 16.5) mm, rotated rx 180 ry 0 rz -180 deg; joints [3.25, 66.553, -28.662, 5.282, -38.009, -4.166]
  Set speed (45.0 mm/s)
  Call Extruder -0.02
  MoveL (T14914) to (104.51, 104.43, 16.5) mm, rotated rx 180 ry 0 rz -180 deg; joints [3.25, 66.553, -28.662, 5.282, -38.009, -4.166]
  Set speed (150.0 mm/s)
  MoveL (T14915) to (104.51, 104.43, 18.5) mm, rotated rx 180 ry 0 rz -180 deg; joints [3.25, 66.553, -28.662, 5.282, -38.009, -4.166]
  MoveL (T14916) to (103.84, 109.5, 18.5) mm, rotated rx 180 ry 0 rz -180 deg; joints [3.25, 66.553, -28.662, 5.282, -38.009, -4.166]
  MoveL (T14917) to (103.84, 109.5, 16.5) mm, rotated rx 180 ry 0 rz -180 deg; joints [3.25, 66.315, -28.622, 5.305, -37.812, -4.196]
  Set speed (40.0 mm/s)
  Call Extruder 2.0
  MoveL (T14918) to (103.84, 109.5, 16.5) mm, rotated rx 180 ry 0 rz -180 deg; joints [1.407, 66.264, -28.527, 2.299, -37.76, -1.818]
  Set speed (36.8 mm/s)
  MoveL (T14919) to (103.84, 109.5, 16.5) mm, rotated rx 180 ry 0 rz -180 deg; joints [1.407, 66.478, -28.563, 2.289, -37.938, -1.806]
  Call Extruder 0.07441
  MoveL (T14920) to (103.84, 111.94, 16.5) mm, rotated rx 180 ry 0 rz -180 deg; joints [1.407, 66.478, -28.563, 2.289, -37.938, -1.806]
  Call Extruder 0.16301
  MoveL (T14921) to (107.63, 108.16, 16.5) mm, rotated rx 180 ry 0 rz -180 deg; joints [1.407, 66.478, -28.563, 2.289, -37.938, -1.806]
  Call Extruder 0.01622
  MoveL (T14922) to (108.16, 108.16, 16.5) mm, rotated rx 180 ry 0 rz -180 deg; joints [1.407, 66.478, -28.563, 2.289, -37.938, -1.806]
  Call Extruder 0.37271
  MoveL (T14923) to (116.81, 116.81, 16.5) mm, rotated rx 180 ry 0 rz -180 deg; joints [1.407, 66.478, -28.563, 2.289, -37.938, -1.806]
  Call Extruder 0.01791
  MoveL (T14924) to (116.81, 117.4, 16.5) mm, rotated rx 180 ry 0 rz -180 deg; joints [1.407, 66.478, -28.563, 2.289, -37.938, -1.806]
  Call Extruder 0.16181
  MoveL (T14925) to (113.06, 121.16, 16.5) mm, rotated rx 180 ry 0 rz -180 deg; joints [1.363, 71.317, -37.664, 2.459, -33.678, -2.047]
  Call Extruder 0.03385
  MoveL (T14926) to (111.94, 121.16, 16.5) mm, rotated rx 180 ry 0 rz -180 deg; joints [1.363, 71.317, -37.664, 2.459, -33.678, -2.047]
  Call Extruder 0.34896
  MoveL (T14927) to (103.84, 113.06, 16.5) mm, rotated rx 180 ry 0 rz -180 deg; joints [3.241, 71.544, -38.091, 5.866, -33.592, -4.891]
  Call Extruder 0.07441
  MoveL (T14928) to (103.84, 115.5, 16.5) mm, rotated rx 180 ry 0 rz -180 deg; joints [3.241, 71.544, -38.091, 5.866, -33.592, -4.891]
  Set speed (45.0 mm/s)
  Call Extruder -1.6
  MoveL (T14929) to (103.84, 115.5, 16.5) mm, rotated rx 180 ry 0 rz -180 deg; joints [3.351, 66.464, -28.536, 5.442, -38.054, -4.29]
  Set speed (120.0 mm/s)
  MoveL (T14930) to (103.84, 115.5, 16.5) mm, rotated rx 180 ry 0 rz -180 deg; joints [3.351, 66.464, -28.536, 5.442, -38.054, -4.29]
  Call Extruder -0.38
  MoveL (T14931) to (103.84, 114.43, 16.5) mm, rotated rx 180 ry 0 rz -180 deg; joints [3.351, 66.464, -28.536, 5.442, -38.054, -4.29]
  Set speed (45.0 mm/s)
  Call Extruder -0.02
  MoveL (T14932) to (103.84, 114.43, 16.5) mm, rotated rx 180 ry 0 rz -180 deg; joints [1.409, 66.273, -28.177, 2.284, -38.118, -1.797]
  Set speed (150.0 mm/s)
  MoveL (T14933) to (103.84, 114.43, 18.5) mm, rotated rx 180 ry 0 rz -180 deg; joints [1.407, 66.463, -28.534, 2.289, -37.951, -1.805]
  MoveL (T14934) to (106.29, 121.16, 18.5) mm, rotated rx 180 ry 0 rz -180 deg; joints [1.407, 66.463, -28.534, 2.289, -37.951, -1.805]
  MoveL (T14935) to (106.29, 121.16, 16.5) mm, rotated rx 180 ry 0 rz -180 deg; joints [1.407, 66.463, -28.534, 2.289, -37.951, -1.805]
  Set speed (40.0 mm/s)
  Call Extruder 2.0
  MoveL (T14936) to (106.29, 121.16, 16.5) mm, rotated rx 180 ry 0 rz -180 deg; joints [1.365, 66.269, -28.169, 2.212, -38.121, -1.741]
  Set speed (36.8 mm/s)
  MoveL (T14937) to (106.29, 121.16, 16.5) mm, rotated rx 180 ry 0 rz -180 deg; joints [1.365, 66.269, -28.169, 2.212, -38.121, -1.741]
  Call Extruder 0.07441
  MoveL (T14938) to (103.84, 121.16, 16.5) mm, rotated rx 180 ry 0 rz -180 deg; joints [1.365, 66.269, -28.169, 2.212, -38.121, -1.741]
  Call Extruder 0.55882
  MoveL (T14939) to (116.81, 108.19, 16.5) mm, rotated rx 180 ry 0 rz -180 deg; joints [1.365, 66.269, -28.169, 2.212, -38.121, -1.741]
  Call Extruder 0.07083
  MoveL (T14940) to (116.81, 110.51, 16.5) mm, rotated rx 180 ry 0 rz -180 deg; joints [1.365, 66.269, -28.169, 2.212, -38.121, -1.741]
  Call Extruder 0.00661
  MoveL (T14941) to (116.9, 110.71, 16.5) mm, rotated rx 180 ry 0 rz -180 deg; joints [1.365, 66.269, -28.169, 2.212, -38.121, -1.741]
  Call Extruder 0.04304
  MoveL (T14942) to (117.9, 111.71, 16.5) mm, rotated rx 180 ry 0 rz -180 deg; joints [1.365, 66.269, -28.169, 2.212, -38.121, -1.741]
  Call Extruder 0.40697
  MoveL (T14943) to (108.45, 121.16, 16.5) mm, rotated rx 180 ry 0 rz -180 deg; joints [1.319, 71.442, -37.899, 2.387, -33.566, -1.989]
  Call Extruder 0.03385
  MoveL (T14944) to (107.34, 121.16, 16.5) mm, rotated rx 180 ry 0 rz -180 deg; joints [1.319, 71.442, -37.899, 2.387, -33.566, -1.989]
  Call Extruder 0.15054
  MoveL (T14945) to (103.84, 117.66, 16.5) mm, rotated rx 180 ry 0 rz -180 deg; joints [1.319, 71.442, -37.899, 2.387, -33.566, -1.989]
  Call Extruder 0.03385
  MoveL (T14946) to (103.84, 116.55, 16.5) mm, rotated rx 180 ry 0 rz -180 deg; joints [3.282, 71.681, -38.348, 5.957, -33.475, -4.974]
  Call Extruder 0.38433
  MoveL (T14947) to (112.77, 107.63, 16.5) mm, rotated rx 180 ry 0 rz -180 deg; joints [3.282, 71.681, -38.348, 5.957, -33.475, -4.974]
  Call Extruder 0.02508
  MoveL (T14948) to (112.18, 107.05, 16.5) mm, rotated rx 180 ry 0 rz -180 deg; joints [3.398, 66.366, -28.351, 5.507, -38.143, -4.336]
  Call Extruder 0.01143
  MoveL (T14949) to (111.92, 107.31, 16.5) mm, rotated rx 180 ry 0 rz -180 deg; joints [3.398, 66.366, -28.351, 5.507, -38.143, -4.336]
  Call Extruder 0.23887
  MoveL (T14950) to (117.46, 112.86, 16.5) mm, rotated rx 180 ry 0 rz -180 deg; joints [1.366, 66.167, -27.977, 2.209, -38.211, -1.736]
  Call Extruder 0.02436
  MoveL (T14951) to (116.9, 113.42, 16.5) mm, rotated rx 180 ry 0 rz -180 deg; joints [1.366, 66.167, -27.977, 2.209, -38.211, -1.736]
  Call Extruder 0.00661
  MoveL (T14952) to (116.81, 113.62, 16.5) mm, rotated rx 180 ry 0 rz -180 deg; joints [1.365, 66.254, -28.14, 2.212, -38.134, -1.74]
  Call Extruder 0.04343
  MoveL (T14953) to (116.81, 115.05, 16.5) mm, rotated rx 180 ry 0 rz -180 deg; joints [1.365, 66.254, -28.14, 2.212, -38.134, -1.74]
  Set speed (45.0 mm/s)
  Call Extruder -1.6
  MoveL (T14954) to (116.81, 115.05, 16.5) mm, rotated rx 180 ry 0 rz -180 deg; joints [1.365, 66.254, -28.14, 2.212, -38.134, -1.74]
  Set speed (120.0 mm/s)
  MoveL (T14955) to (116.81, 115.05, 16.5) mm, rotated rx 180 ry 0 rz -180 deg; joints [1.332, 66.062, -27.779, 2.15, -38.302, -1.688]
  Call Extruder -0.38
  MoveL (T14956) to (116.81, 113.98, 16.5) mm, rotated rx 180 ry 0 rz -180 deg; joints [1.332, 66.062, -27.779, 2.15, -38.302, -1.688]
  Set speed (45.0 mm/s)
  Call Extruder -0.02
  MoveL (T14957) to (116.81, 113.98, 16.5) mm, rotated rx 180 ry 0 rz -180 deg; joints [1.332, 66.062, -27.779, 2.15, -38.302, -1.688]
  Set speed (150.0 mm/s)
  MoveL (T14958) to (116.81, 113.98, 18.5) mm, rotated rx 180 ry 0 rz -180 deg; joints [1.332, 66.062, -27.779, 2.15, -38.302, -1.688]
  MoveL (T14959) to (104.34, 103.54, 18.5) mm, rotated rx 180 ry 0 rz -180 deg; joints [1.332, 66.062, -27.779, 2.15, -38.302, -1.688]
  MoveL (T14960) to (104.34, 103.54, 16.7) mm, rotated rx 180 ry 0 rz -180 deg; joints [1.332, 66.062, -27.779, 2.15, -38.302, -1.688]
  Set speed (40.0 mm/s)
  Call Extruder 2.0
  MoveL (T14961) to (104.34, 103.54, 16.7) mm, rotated rx 180 ry 0 rz -180 deg; joints [1.323, 66.061, -27.778, 2.135, -38.302, -1.676]
  Set speed (37.7 mm/s)
  MoveL (T14962) to (104.34, 103.54, 16.7) mm, rotated rx 180 ry 0 rz -180 deg; joints [1.276, 71.568, -38.136, 2.315, -33.454, -1.932]
  Call Extruder 0.52159
  MoveL (T14963) to (121.46, 103.54, 16.7) mm, rotated rx 180 ry 0 rz -180 deg; joints [1.276, 71.568, -38.136, 2.315, -33.454, -1.932]
  Call Extruder 0.54596
  MoveL (T14964) to (121.46, 121.46, 16.7) mm, rotated rx 180 ry 0 rz -180 deg; joints [3.322, 71.818, -38.607, 6.048, -33.358, -5.058]
  Call Extruder 0.54596
  MoveL (T14965) to (103.54, 121.46, 16.7) mm, rotated rx 180 ry 0 rz -180 deg; joints [3.322, 71.818, -38.607, 6.048, -33.358, -5.058]
  Call Extruder 0.54596
  MoveL (T14966) to (103.54, 103.54, 16.7) mm, rotated rx 180 ry 0 rz -180 deg; joints [3.322, 71.818, -38.607, 6.048, -33.358, -5.058]
  Call Extruder 0.02254
  MoveL (T14967) to (104.28, 103.54, 16.7) mm, rotated rx 180 ry 0 rz -180 deg; joints [3.445, 66.268, -28.167, 5.571, -38.233, -4.382]
  Set speed (150.0 mm/s)
  MoveL (T14968) to (103.53, 103.13, 16.7) mm, rotated rx 180 ry 0 rz -180 deg; joints [3.445, 66.268, -28.167, 5.571, -38.233, -4.382]
  Set speed (37.7 mm/s)
  MoveL (T14969) to (103.53, 103.13, 16.7) mm, rotated rx 180 ry 0 rz -180 deg; joints [3.445, 66.268, -28.167, 5.571, -38.233, -4.382]
  Call Extruder 0.55858
  MoveL (T14970) to (121.87, 103.13, 16.7) mm, rotated rx 180 ry 0 rz -180 deg; joints [1.339, 66.062, -27.78, 2.161, -38.302, -1.696]
  Call Extruder 0.57077
  MoveL (T14971) to (121.87, 121.87, 16.7) mm, rotated rx 180 ry 0 rz -180 deg; joints [1.339, 66.062, -27.78, 2.161, -38.302, -1.696]
  Call Extruder 0.57077
  MoveL (T14972) to (103.13, 121.87, 16.7) mm, rotated rx 180 ry 0 rz -180 deg; joints [1.326, 66.077, -27.807, 2.14, -38.289, -1.68]
  Call Extruder 0.57077
  MoveL (T14973) to (103.13, 103.13, 16.7) mm, rotated rx 180 ry 0 rz -180 deg; joints [1.326, 66.077, -27.807, 2.14, -38.289, -1.68]
  Call Extruder 0.01036
  MoveL (T14974) to (103.47, 103.13, 16.7) mm, rotated rx 180 ry 0 rz -180 deg; joints [1.326, 66.077, -27.807, 2.14, -38.289, -1.68]
  Set speed (150.0 mm/s)
  MoveL (T14975) to (102.72, 102.81, 16.7) mm, rotated rx 180 ry 0 rz -180 deg; joints [1.326, 66.077, -27.807, 2.14, -38.289, -1.68]
  Set speed (25.0 mm/s)
  MoveL (T14976) to (102.72, 102.81, 16.7) mm, rotated rx 180 ry 0 rz -180 deg; joints [1.326, 66.077, -27.807, 2.14, -38.289, -1.68]
  Call Extruder 0.00259
  MoveL (T14977) to (102.72, 102.72, 16.7) mm, rotated rx 180 ry 0 rz -180 deg; joints [1.326, 66.077, -27.807, 2.14, -38.289, -1.68]
  Call Extruder 0.59557
  MoveL (T14978) to (122.28, 102.72, 16.7) mm, rotated rx 180 ry 0 rz -180 deg; joints [1.326, 66.077, -27.807, 2.14, -38.289, -1.68]
  Call Extruder 0.59557
  MoveL (T14979) to (122.28, 122.28, 16.7) mm, rotated rx 180 ry 0 rz -180 deg; joints [1.326, 66.077, -27.807, 2.14, -38.289, -1.68]
  Call Extruder 0.59557
  MoveL (T14980) to (102.72, 122.28, 16.7) mm, rotated rx 180 ry 0 rz -180 deg; joints [1.326, 66.077, -27.807, 2.14, -38.289, -1.68]
  Call Extruder 0.59115
  MoveL (T14981) to (102.72, 102.87, 16.7) mm, rotated rx 180 ry 0 rz -180 deg; joints [1.323, 66.061, -27.778, 2.135, -38.302, -1.676]
  Set speed (150.0 mm/s)
  MoveL (T14982) to (102.78, 102.75, 16.7) mm, rotated rx 180 ry 0 rz -180 deg; joints [1.323, 66.061, -27.778, 2.135, -38.302, -1.676]
  Set speed (45.0 mm/s)
  Call Extruder -1.6
  MoveL (T14983) to (102.78, 102.75, 16.7) mm, rotated rx 180 ry 0 rz -180 deg; joints [1.323, 66.061, -27.778, 2.135, -38.302, -1.676]
  Set speed (120.0 mm/s)
  MoveL (T14984) to (102.78, 102.75, 16.7) mm, rotated rx 180 ry 0 rz -180 deg; joints [1.321, 66.296, -28.22, 2.141, -38.096, -1.685]
  Call Extruder -0.05166
  MoveL (T14985) to (102.72, 102.72, 16.7) mm, rotated rx 180 ry 0 rz -180 deg; joints [1.321, 66.296, -28.22, 2.141, -38.096, -1.685]
  Call Extruder -0.32834
  MoveL (T14986) to (103.65, 102.72, 16.7) mm, rotated rx 180 ry 0 rz -180 deg; joints [1.321, 66.296, -28.22, 2.141, -38.096, -1.685]
  Set speed (45.0 mm/s)
  Call Extruder -0.02
  MoveL (T14987) to (103.65, 102.72, 16.7) mm, rotated rx 180 ry 0 rz -180 deg; joints [1.321, 66.296, -28.22, 2.141, -38.096, -1.685]
  Set speed (150.0 mm/s)
  MoveL (T14988) to (103.65, 102.72, 18.7) mm, rotated rx 180 ry 0 rz -180 deg; joints [1.321, 66.296, -28.22, 2.141, -38.096, -1.685]
  MoveL (T14989) to (103.84, 106.29, 18.7) mm, rotated rx 180 ry 0 rz -180 deg; joints [1.321, 66.296, -28.22, 2.141, -38.096, -1.685]
  MoveL (T14990) to (103.84, 106.29, 16.7) mm, rotated rx 180 ry 0 rz -180 deg; joints [1.321, 66.296, -28.22, 2.141, -38.096, -1.685]
  Set speed (40.0 mm/s)
  Call Extruder 2.0
  MoveL (T14991) to (103.84, 106.29, 16.7) mm, rotated rx 180 ry 0 rz -180 deg; joints [3.142, 71.254, -37.94, 5.708, -33.445, -4.768]
  Set speed (37.7 mm/s)
  MoveL (T14992) to (103.84, 106.29, 16.7) mm, rotated rx 180 ry 0 rz -180 deg; joints [3.142, 71.489, -37.987, 5.68, -33.632, -4.734]
  Call Extruder 0.07441
  MoveL (T14993) to (103.84, 103.84, 16.7) mm, rotated rx 180 ry 0 rz -180 deg; joints [3.142, 71.489, -37.987, 5.68, -33.632, -4.734]
  Call Extruder 0.0111
  MoveL (T14994) to (104.1, 104.1, 16.7) mm, rotated rx 180 ry 0 rz -180 deg; joints [3.142, 71.489, -37.987, 5.68, -33.632, -4.734]
  Call Extruder 0.05294
  MoveL (T14995) to (104.1, 105.84, 16.7) mm, rotated rx 180 ry 0 rz -180 deg; joints [3.142, 71.489, -37.987, 5.68, -33.632, -4.734]
  Call Extruder 0.00661
  MoveL (T14996) to (104.18, 106.04, 16.7) mm, rotated rx 180 ry 0 rz -180 deg; joints [3.142, 71.489, -37.987, 5.68, -33.632, -4.734]
  Call Extruder 0.02065
  MoveL (T14997) to (104.66, 106.52, 16.7) mm, rotated rx 180 ry 0 rz -180 deg; joints [3.142, 71.489, -37.987, 5.68, -33.632, -4.734]
  Call Extruder 0.03528
  MoveL (T14998) to (103.84, 107.34, 16.7) mm, rotated rx 180 ry 0 rz -180 deg; joints [3.214, 71.296, -37.625, 5.783, -33.807, -4.81]
  Call Extruder 0.03385
  MoveL (T14999) to (103.84, 108.45, 16.7) mm, rotated rx 180 ry 0 rz -180 deg; joints [3.214, 71.296, -37.625, 5.783, -33.807, -4.81]
  Call Extruder 0.54738
  MoveL (T15000) to (116.55, 121.16, 16.7) mm, rotated rx 180 ry 0 rz -180 deg; joints [3.217, 71.115, -37.284, 5.765, -33.966, -4.787]
  Call Extruder 0.03385
  MoveL (T15001) to (117.66, 121.16, 16.7) mm, rotated rx 180 ry 0 rz -180 deg; joints [3.217, 71.115, -37.284, 5.765, -33.966, -4.787]
  Call Extruder 0.0423
  MoveL (T15002) to (118.64, 120.17, 16.7) mm, rotated rx 180 ry 0 rz -180 deg; joints [3.217, 71.115, -37.284, 5.765, -33.966, -4.787]
  Call Extruder 0.01225
  MoveL (T15003) to (118.93, 120.46, 16.7) mm, rotated rx 180 ry 0 rz -180 deg; joints [3.102, 71.424, -37.865, 5.599, -33.685, -4.663]
  Call Extruder 0.00661
  MoveL (T15004) to (119.13, 120.54, 16.7) mm, rotated rx 180 ry 0 rz -180 deg; joints [3.102, 71.424, -37.865, 5.599, -33.685, -4.663]
  Call Extruder 0.04314
  MoveL (T15005) to (120.54, 120.54, 16.7) mm, rotated rx 180 ry 0 rz -180 deg; joints [3.102, 71.424, -37.865, 5.599, -33.685, -4.663]
  Call Extruder 0.02637
  MoveL (T15006) to (121.16, 121.16, 16.7) mm, rotated rx 180 ry 0 rz -180 deg; joints [3.041, 71.414, -37.847, 5.488, -33.689, -4.571]
  Call Extruder 0.07441
  MoveL (T15007) to (118.71, 121.16, 16.7) mm, rotated rx 180 ry 0 rz -180 deg; joints [3.041, 71.414, -37.847, 5.488, -33.689, -4.571]
  Set speed (45.0 mm/s)
  Call Extruder -1.6
  MoveL (T15008) to (118.71, 121.16, 16.7) mm, rotated rx 180 ry 0 rz -180 deg; joints [3.041, 71.414, -37.847, 5.488, -33.689, -4.571]
  Set speed (120.0 mm/s)
  MoveL (T15009) to (118.71, 121.16, 16.7) mm, rotated rx 180 ry 0 rz -180 deg; joints [3.221, 70.936, -36.946, 5.748, -34.123, -4.763]
  Call Extruder -0.38
  MoveL (T15010) to (119.78, 121.16, 16.7) mm, rotated rx 180 ry 0 rz -180 deg; joints [3.221, 70.936, -36.946, 5.748, -34.123, -4.763]
  Set speed (45.0 mm/s)
  Call Extruder -0.02
  MoveL (T15011) to (119.78, 121.16, 16.7) mm, rotated rx 180 ry 0 rz -180 deg; joints [3.221, 70.936, -36.946, 5.748, -34.123, -4.763]
  Set speed (150.0 mm/s)
  MoveL (T15012) to (119.78, 121.16, 18.7) mm, rotated rx 180 ry 0 rz -180 deg; joints [3.224, 70.758, -36.611, 5.731, -34.28, -4.741]
  MoveL (T15013) to (116.81, 115.05, 18.7) mm, rotated rx 180 ry 0 rz -180 deg; joints [3.224, 70.758, -36.611, 5.731, -34.28, -4.741]
  MoveL (T15014) to (116.81, 115.05, 16.7) mm, rotated rx 180 ry 0 rz -180 deg; joints [2.98, 71.405, -37.829, 5.377, -33.693, -4.478]
  Set speed (40.0 mm/s)
  Call Extruder 2.0
  MoveL (T15015) to (116.81, 115.05, 16.7) mm, rotated rx 180 ry 0 rz -180 deg; joints [2.98, 71.405, -37.829, 5.377, -33.693, -4.478]
  Set speed (37.7 mm/s)
  MoveL (T15016) to (116.81, 115.05, 16.7) mm, rotated rx 180 ry 0 rz -180 deg; joints [2.98, 71.405, -37.829, 5.377, -33.693, -4.478]
  Call Extruder 0.04343
  MoveL (T15017) to (116.81, 113.62, 16.7) mm, rotated rx 180 ry 0 rz -180 deg; joints [2.919, 71.395, -37.811, 5.267, -33.696, -4.386]
  Call Extruder 0.00661
  MoveL (T15018) to (116.9, 113.42, 16.7) mm, rotated rx 180 ry 0 rz -180 deg; joints [2.919, 71.395, -37.811, 5.267, -33.696, -4.386]
  Call Extruder 0.02436
  MoveL (T15019) to (117.46, 112.86, 16.7) mm, rotated rx 180 ry 0 rz -180 deg; joints [2.919, 71.395, -37.811, 5.267, -33.696, -4.386]
  Call Extruder 0.23887
  MoveL (T15020) to (111.92, 107.31, 16.7) mm, rotated rx 180 ry 0 rz -180 deg; joints [3.228, 70.581, -36.279, 5.714, -34.435, -4.718]
  Call Extruder 0.01143
  MoveL (T15021) to (112.18, 107.05, 16.7) mm, rotated rx 180 ry 0 rz -180 deg; joints [3.228, 70.581, -36.279, 5.714, -34.435, -4.718]
  Call Extruder 0.02508
  MoveL (T15022) to (112.77, 107.63, 16.7) mm, rotated rx 180 ry 0 rz -180 deg; joints [3.228, 70.581, -36.279, 5.714, -34.435, -4.718]
  Call Extruder 0.38433
  MoveL (T15023) to (103.84, 116.55, 16.7) mm, rotated rx 180 ry 0 rz -180 deg; joints [3.231, 70.406, -35.949, 5.698, -34.589, -4.696]
  Call Extruder 0.03385
  MoveL (T15024) to (103.84, 117.66, 16.7) mm, rotated rx 180 ry 0 rz -180 deg; joints [3.231, 70.406, -35.949, 5.698, -34.589, -4.696]
  Call Extruder 0.15054
  MoveL (T15025) to (107.34, 121.16, 16.7) mm, rotated rx 180 ry 0 rz -180 deg; joints [3.231, 70.406, -35.949, 5.698, -34.589, -4.696]
  Call Extruder 0.03385
  MoveL (T15026) to (108.45, 121.16, 16.7) mm, rotated rx 180 ry 0 rz -180 deg; joints [2.858, 71.386, -37.794, 5.157, -33.7, -4.294]
  Call Extruder 0.40697
  MoveL (T15027) to (117.9, 111.71, 16.7) mm, rotated rx 180 ry 0 rz -180 deg; joints [2.858, 71.386, -37.794, 5.157, -33.7, -4.294]
  Call Extruder 0.04304
  MoveL (T15028) to (116.9, 110.71, 16.7) mm, rotated rx 180 ry 0 rz -180 deg; joints [2.858, 71.386, -37.794, 5.157, -33.7, -4.294]
  Call Extruder 0.00661
  MoveL (T15029) to (116.81, 110.51, 16.7) mm, rotated rx 180 ry 0 rz -180 deg; joints [2.797, 71.377, -37.777, 5.046, -33.703, -4.201]
  Call Extruder 0.07083
  MoveL (T15030) to (116.81, 108.19, 16.7) mm, rotated rx 180 ry 0 rz -180 deg; joints [2.797, 71.377, -37.777, 5.046, -33.703, -4.201]
  Call Extruder 0.55882
  MoveL (T15031) to (103.84, 121.16, 16.7) mm, rotated rx 180 ry 0 rz -180 deg; joints [2.797, 71.377, -37.777, 5.046, -33.703, -4.201]
  Call Extruder 0.07441
  MoveL (T15032) to (106.29, 121.16, 16.7) mm, rotated rx 180 ry 0 rz -180 deg; joints [3.235, 70.232, -35.622, 5.682, -34.742, -4.674]
  Set speed (45.0 mm/s)
  Call Extruder -1.6
  MoveL (T15033) to (106.29, 121.16, 16.7) mm, rotated rx 180 ry 0 rz -180 deg; joints [3.235, 70.232, -35.622, 5.682, -34.742, -4.674]
  Set speed (120.0 mm/s)
  MoveL (T15034) to (106.29, 121.16, 16.7) mm, rotated rx 180 ry 0 rz -180 deg; joints [3.235, 70.232, -35.622, 5.682, -34.742, -4.674]
  Call Extruder -0.38
  MoveL (T15035) to (105.22, 121.16, 16.7) mm, rotated rx 180 ry 0 rz -180 deg; joints [3.238, 70.059, -35.297, 5.667, -34.894, -4.653]
  Set speed (45.0 mm/s)
  Call Extruder -0.02
  MoveL (T15036) to (105.22, 121.16, 16.7) mm, rotated rx 180 ry 0 rz -180 deg; joints [2.737, 71.368, -37.76, 4.936, -33.706, -4.109]
  Set speed (150.0 mm/s)
  MoveL (T15037) to (105.22, 121.16, 18.7) mm, rotated rx 180 ry 0 rz -180 deg; joints [2.676, 71.36, -37.744, 4.825, -33.71, -4.017]
  MoveL (T15038) to (103.84, 115.5, 18.7) mm, rotated rx 180 ry 0 rz -180 deg; joints [2.676, 71.36, -37.744, 4.825, -33.71, -4.017]
  MoveL (T15039) to (103.84, 115.5, 16.7) mm, rotated rx 180 ry 0 rz -180 deg; joints [2.676, 71.36, -37.744, 4.825, -33.71, -4.017]
  Set speed (40.0 mm/s)
  Call Extruder 2.0
  MoveL (T15040) to (103.84, 115.5, 16.7) mm, rotated rx 180 ry 0 rz -180 deg; joints [3.242, 69.888, -34.974, 5.651, -35.044, -4.632]
  Set speed (37.7 mm/s)
  MoveL (T15041) to (103.84, 115.5, 16.7) mm, rotated rx 180 ry 0 rz -180 deg; joints [3.242, 69.888, -34.974, 5.651, -35.044, -4.632]
  Call Extruder 0.07441
  MoveL (T15042) to (103.84, 113.06, 16.7) mm, rotated rx 180 ry 0 rz -180 deg; joints [3.242, 69.888, -34.974, 5.651, -35.044, -4.632]
  Call Extruder 0.34896
  MoveL (T15043) to (111.94, 121.16, 16.7) mm, rotated rx 180 ry 0 rz -180 deg; joints [3.245, 69.717, -34.654, 5.636, -35.194, -4.611]
  Call Extruder 0.03385
  MoveL (T15044) to (113.06, 121.16, 16.7) mm, rotated rx 180 ry 0 rz -180 deg; joints [3.245, 69.717, -34.654, 5.636, -35.194, -4.611]
  Call Extruder 0.16181
  MoveL (T15045) to (116.81, 117.4, 16.7) mm, rotated rx 180 ry 0 rz -180 deg; joints [2.615, 71.351, -37.728, 4.715, -33.713, -3.925]
  Call Extruder 0.01791
  MoveL (T15046) to (116.81, 116.81, 16.7) mm, rotated rx 180 ry 0 rz -180 deg; joints [2.615, 71.351, -37.728, 4.715, -33.713, -3.925]
  Call Extruder 0.37271
  MoveL (T15047) to (108.16, 108.16, 16.7) mm, rotated rx 180 ry 0 rz -180 deg; joints [2.615, 71.351, -37.728, 4.715, -33.713, -3.925]
  Call Extruder 0.01622
  MoveL (T15048) to (107.63, 108.16, 16.7) mm, rotated rx 180 ry 0 rz -180 deg; joints [2.554, 71.343, -37.713, 4.604, -33.716, -3.833]
  Call Extruder 0.16301
  MoveL (T15049) to (103.84, 111.94, 16.7) mm, rotated rx 180 ry 0 rz -180 deg; joints [2.554, 71.343, -37.713, 4.604, -33.716, -3.833]
  Call Extruder 0.07441
  MoveL (T15050) to (103.84, 109.5, 16.7) mm, rotated rx 180 ry 0 rz -180 deg; joints [2.554, 71.343, -37.713, 4.604, -33.716, -3.833]
  Set speed (45.0 mm/s)
  Call Extruder -1.6
  MoveL (T15051) to (103.84, 109.5, 16.7) mm, rotated rx 180 ry 0 rz -180 deg; joints [3.249, 69.548, -34.336, 5.622, -35.342, -4.591]
  Set speed (120.0 mm/s)
  MoveL (T15052) to (103.84, 109.5, 16.7) mm, rotated rx 180 ry 0 rz -180 deg; joints [3.252, 69.381, -34.021, 5.608, -35.49, -4.571]
  Call Extruder -0.38
  MoveL (T15053) to (103.84, 110.57, 16.7) mm, rotated rx 180 ry 0 rz -180 deg; joints [3.252, 69.381, -34.021, 5.608, -35.49, -4.571]
  Set speed (45.0 mm/s)
  Call Extruder -0.02
  MoveL (T15054) to (103.84, 110.57, 16.7) mm, rotated rx 180 ry 0 rz -180 deg; joints [3.252, 69.381, -34.021, 5.608, -35.49, -4.571]
  Set speed (150.0 mm/s)
  MoveL (T15055) to (103.84, 110.57, 18.7) mm, rotated rx 180 ry 0 rz -180 deg; joints [2.493, 71.335, -37.697, 4.494, -33.719, -3.74]
  MoveL (T15056) to (121.34, 104.69, 18.7) mm, rotated rx 180 ry 0 rz -180 deg; joints [2.432, 71.327, -37.683, 4.384, -33.722, -3.648]
  MoveL (T15057) to (121.34, 104.69, 16.7) mm, rotated rx 180 ry 0 rz -180 deg; joints [2.432, 71.327, -37.683, 4.384, -33.722, -3.648]
  Set speed (40.0 mm/s)
  Call Extruder 2.0
  MoveL (T15058) to (121.34, 104.69, 16.7) mm, rotated rx 180 ry 0 rz -180 deg; joints [3.256, 69.214, -33.707, 5.593, -35.636, -4.551]
  Set speed (37.7 mm/s)
  MoveL (T15059) to (121.34, 104.69, 16.7) mm, rotated rx 180 ry 0 rz -180 deg; joints [3.259, 69.048, -33.396, 5.58, -35.781, -4.531]
  Call Extruder 0.03095
  MoveL (T15060) to (120.62, 103.98, 16.7) mm, rotated rx 180 ry 0 rz -180 deg; joints [3.259, 69.048, -33.396, 5.58, -35.781, -4.531]
  Call Extruder 0.01768
  MoveL (T15061) to (120.05, 103.98, 16.7) mm, rotated rx 180 ry 0 rz -180 deg; joints [3.259, 69.048, -33.396, 5.58, -35.781, -4.531]
  Call Extruder 0.04803
  MoveL (T15062) to (121.16, 105.09, 16.7) mm, rotated rx 180 ry 0 rz -180 deg; joints [2.371, 71.319, -37.668, 4.274, -33.725, -3.556]
  Call Extruder 0.01769
  MoveL (T15063) to (121.16, 105.67, 16.7) mm, rotated rx 180 ry 0 rz -180 deg; joints [2.371, 71.319, -37.668, 4.274, -33.725, -3.556]
  Call Extruder 0.07889
  MoveL (T15064) to (119.33, 103.84, 16.7) mm, rotated rx 180 ry 0 rz -180 deg; joints [2.31, 71.312, -37.654, 4.163, -33.728, -3.464]
  Call Extruder 0.01769
  MoveL (T15065) to (118.75, 103.84, 16.7) mm, rotated rx 180 ry 0 rz -180 deg; joints [3.263, 68.884, -33.087, 5.566, -35.926, -4.512]
  Call Extruder 0.10391
  MoveL (T15066) to (121.16, 106.25, 16.7) mm, rotated rx 180 ry 0 rz -180 deg; joints [3.263, 68.884, -33.087, 5.566, -35.926, -4.512]
  Call Extruder 0.01769
  MoveL (T15067) to (121.16, 106.82, 16.7) mm, rotated rx 180 ry 0 rz -180 deg; joints [3.266, 68.721, -32.78, 5.553, -36.069, -4.493]
  Call Extruder 0.12893
  MoveL (T15068) to (118.18, 103.84, 16.7) mm, rotated rx 180 ry 0 rz -180 deg; joints [3.266, 68.721, -32.78, 5.553, -36.069, -4.493]
  Call Extruder 0.01769
  MoveL (T15069) to (117.6, 103.84, 16.7) mm, rotated rx 180 ry 0 rz -180 deg; joints [2.249, 71.305, -37.641, 4.053, -33.73, -3.373]
  Call Extruder 0.15395
  MoveL (T15070) to (121.16, 107.4, 16.7) mm, rotated rx 180 ry 0 rz -180 deg; joints [2.249, 71.305, -37.641, 4.053, -33.73, -3.373]
  Call Extruder 0.01769
  MoveL (T15071) to (121.16, 107.98, 16.7) mm, rotated rx 180 ry 0 rz -180 deg; joints [2.249, 71.305, -37.641, 4.053, -33.73, -3.373]
  Call Extruder 0.17896
  MoveL (T15072) to (117.02, 103.84, 16.7) mm, rotated rx 180 ry 0 rz -180 deg; joints [2.188, 71.298, -37.627, 3.943, -33.733, -3.281]
  Call Extruder 0.01769
  MoveL (T15073) to (116.44, 103.84, 16.7) mm, rotated rx 180 ry 0 rz -180 deg; joints [2.188, 71.298, -37.627, 3.943, -33.733, -3.281]
  Call Extruder 0.20398
  MoveL (T15074) to (121.16, 108.56, 16.7) mm, rotated rx 180 ry 0 rz -180 deg; joints [2.188, 71.298, -37.627, 3.943, -33.733, -3.281]
  Call Extruder 0.01769
  MoveL (T15075) to (121.16, 109.14, 16.7) mm, rotated rx 180 ry 0 rz -180 deg; joints [3.27, 68.559, -32.475, 5.54, -36.212, -4.475]
  Call Extruder 0.229
  MoveL (T15076) to (115.86, 103.84, 16.7) mm, rotated rx 180 ry 0 rz -180 deg; joints [3.273, 68.397, -32.172, 5.527, -36.353, -4.457]
  Call Extruder 0.01769
  MoveL (T15077) to (115.28, 103.84, 16.7) mm, rotated rx 180 ry 0 rz -180 deg; joints [3.273, 68.397, -32.172, 5.527, -36.353, -4.457]
  Call Extruder 0.25402
  MoveL (T15078) to (121.16, 109.72, 16.7) mm, rotated rx 180 ry 0 rz -180 deg; joints [2.127, 71.291, -37.614, 3.833, -33.736, -3.189]
  Call Extruder 0.01769
  MoveL (T15079) to (121.16, 110.29, 16.7) mm, rotated rx 180 ry 0 rz -180 deg; joints [2.127, 71.291, -37.614, 3.833, -33.736, -3.189]
  Call Extruder 0.27904
  MoveL (T15080) to (114.71, 103.84, 16.7) mm, rotated rx 180 ry 0 rz -180 deg; joints [2.067, 71.284, -37.602, 3.723, -33.738, -3.097]
  Call Extruder 0.01769
  MoveL (T15081) to (114.13, 103.84, 16.7) mm, rotated rx 180 ry 0 rz -180 deg; joints [2.067, 71.284, -37.602, 3.723, -33.738, -3.097]
  Call Extruder 0.30406
  MoveL (T15082) to (121.16, 110.87, 16.7) mm, rotated rx 180 ry 0 rz -180 deg; joints [2.067, 71.284, -37.602, 3.723, -33.738, -3.097]
  Call Extruder 0.01769
  MoveL (T15083) to (121.16, 111.45, 16.7) mm, rotated rx 180 ry 0 rz -180 deg; joints [3.277, 68.238, -31.871, 5.515, -36.494, -4.438]
  Call Extruder 0.32908
  MoveL (T15084) to (113.55, 103.84, 16.7) mm, rotated rx 180 ry 0 rz -180 deg; joints [3.277, 68.238, -31.871, 5.515, -36.494, -4.438]
  Call Extruder 0.01769
  MoveL (T15085) to (112.97, 103.84, 16.7) mm, rotated rx 180 ry 0 rz -180 deg; joints [3.28, 68.078, -31.572, 5.503, -36.634, -4.421]
  Call Extruder 0.3541
  MoveL (T15086) to (121.16, 112.03, 16.7) mm, rotated rx 180 ry 0 rz -180 deg; joints [3.28, 68.078, -31.572, 5.503, -36.634, -4.421]
  Call Extruder 0.01769
  MoveL (T15087) to (121.16, 112.61, 16.7) mm, rotated rx 180 ry 0 rz -180 deg; joints [2.006, 71.278, -37.59, 3.613, -33.741, -3.005]
  Call Extruder 0.1702
  MoveL (T15088) to (117.22, 108.67, 16.7) mm, rotated rx 180 ry 0 rz -180 deg; joints [2.006, 71.278, -37.59, 3.613, -33.741, -3.005]
  Call Extruder 0.01768
  MoveL (T15089) to (117.22, 109.25, 16.7) mm, rotated rx 180 ry 0 rz -180 deg; joints [1.945, 71.271, -37.578, 3.503, -33.743, -2.914]
